// TwinCAT 3 PLC project PLC
// ProgramVersion: 3.1.4024.0
// libraries:
//   EfficientIO Energy Basic, * (EfficientIO)
//   Lynus Persistent Data V1, * (Lynus AG)
//   Lynus Standards, * (EfficientIO)
//   Tc2_EtherCAT, * (Beckhoff Automation GmbH)
//   Tc2_Standard, * (Beckhoff Automation GmbH)
//   Tc2_System, * (Beckhoff Automation GmbH)
//   Tc2_Utilities, * (Beckhoff Automation GmbH)
//   Tc3_Module, * (Beckhoff Automation GmbH)
// project tree:
//   FBs/EL3443_DPM/DUTs/ E_EL3443_DPM_Phase.TcDUT (not stored), E_EL3443_DPM_Total.TcDUT (not stored), MDP5001_341_7CD731EE.TcDUT (not stored), MDP5001_341_I_7CD731EE.TcDUT (not stored), MDP5001_341_O_7CD731EE.TcDUT (not stored), ST_EL3443_DPM_MUX_REAL.TcDUT (not stored), ST_EL3443_DPM_MUX_ULINT.TcDUT (not stored), ST_EL3443_DPM_StatusLx.TcDUT (not stored), ST_EL3443_DPM_StatusTotal.TcDUT (not stored), ST_EL3443_DPM_VariantLx.TcDUT (not stored), ST_EL3443_DPM_VariantTotal.TcDUT (not stored), ST_EL3443_DPM_VariantValues.TcDUT (not stored)
//   FBs/EL3443_DPM/ FB_EL3443_DPM.TcPOU (not stored)
//   FBs/EL3446 FW02 or higher/DUTs/ E_EL3446_Phase.TcDUT (not stored), MDP5001_342_066CA8C6.TcDUT (not stored), MDP5001_342_I_066CA8C6.TcDUT (not stored), MDP5001_342_O_066CA8C6.TcDUT (not stored), ST_EL3446_MUX_REAL.TcDUT, ST_EL3446_MUX_ULINT.TcDUT (not stored), ST_EL3446_StatusIx.TcDUT (not stored), ST_EL3446_VariantIx.TcDUT (not stored), ST_EL3446_VariantValues.TcDUT (not stored)
//   FBs/EL3446 FW02 or higher/ FB_EL3446.TcPOU (not stored)
//   FBs/ FB_CoE_EL3443.TcPOU (not stored), FB_CoE_EL3446.TcPOU (not stored), FB_EM_Beckhoff_EL3443.TcPOU (not stored), FB_EM_Beckhoff_EL3446.TcPOU (not stored)
//   / PlcTask.TcTTO
//   POUs/ prgEM.TcPOU, prgHW.TcPOU
// real-time tasks:
//   TASK PlcTask: cycle T#10ms, priority 20, ADS port 350
// I/O:
//   DEVICE Gerät 2 (EtherCAT), AmsNetId 5.146.125.98.3.1
//     Klemme 1 (EK1200) [EK1200-5000 EtherCAT Netzteil (2A E-Bus)]
//       Klemme 2 (EL3443) [EL3443 3K. Leistungsmessung]
//       Klemme 3 (EL3446) [EL3446 DPM 6 K. Strommessklemme]
//       Klemme 4 (EL3446) [EL3446 DPM 6 K. Strommessklemme]
//       Klemme 5 (EL9011) [EL9011 Endklemme]
// variable links:
//   PLC/PLC Instance <-> Device 2 (EtherCAT)/Term 1 (EK1200)/Term 2 (EL3443)
//     PlcTask Inputs/prgHW.MDP5001_341_DPM_Data_Data_{1..20} <-> DPM Data/Data {1..20}  (20 links)
//     PlcTask Inputs/prgHW.MDP5001_341_L1_Basic_Current <-> L1 Basic/Current
//     PlcTask Inputs/prgHW.MDP5001_341_L2_Basic_Current <-> L2 Basic/Current
//     PlcTask Inputs/prgHW.MDP5001_341_L3_Basic_Current <-> L3 Basic/Current
//     PlcTask Inputs/prgHW.MDP5001_341_L1_Basic_Voltage <-> L1 Basic/Voltage
//     PlcTask Inputs/prgHW.MDP5001_341_L2_Basic_Voltage <-> L2 Basic/Voltage
//     PlcTask Inputs/prgHW.MDP5001_341_L3_Basic_Voltage <-> L3 Basic/Voltage
//     PlcTask Inputs/prgHW.MDP5001_341_L1_Power_Active_Power <-> L1 Power/Active Power
//     PlcTask Inputs/prgHW.MDP5001_341_L2_Power_Active_Power <-> L2 Power/Active Power
//     PlcTask Inputs/prgHW.MDP5001_341_L3_Power_Active_Power <-> L3 Power/Active Power
//     PlcTask Inputs/prgHW.MDP5001_341_L1_Power_Apparent_Power <-> L1 Power/Apparent Power
//     PlcTask Inputs/prgHW.MDP5001_341_L2_Power_Apparent_Power <-> L2 Power/Apparent Power
//     PlcTask Inputs/prgHW.MDP5001_341_L3_Power_Apparent_Power <-> L3 Power/Apparent Power
//     PlcTask Inputs/prgHW.MDP5001_341_L1_Power_Power_Factor <-> L1 Power/Power Factor
//     PlcTask Inputs/prgHW.MDP5001_341_L2_Power_Power_Factor <-> L2 Power/Power Factor
//     PlcTask Inputs/prgHW.MDP5001_341_L3_Power_Power_Factor <-> L3 Power/Power Factor
//     PlcTask Inputs/prgHW.MDP5001_341_L1_Power_Reactive_Power <-> L1 Power/Reactive Power
//     PlcTask Inputs/prgHW.MDP5001_341_L2_Power_Reactive_Power <-> L2 Power/Reactive Power
//     PlcTask Inputs/prgHW.MDP5001_341_L3_Power_Reactive_Power <-> L3 Power/Reactive Power
//     PlcTask Inputs/prgHW.MDP5001_341_L1_Status_Current_Guard_Error <-> L1 Status/Current Guard Error
//     PlcTask Inputs/prgHW.MDP5001_341_L2_Status_Current_Guard_Error <-> L2 Status/Current Guard Error
//     PlcTask Inputs/prgHW.MDP5001_341_L3_Status_Current_Guard_Error <-> L3 Status/Current Guard Error
//     PlcTask Inputs/prgHW.MDP5001_341_L1_Status_Current_Guard_Warning <-> L1 Status/Current Guard Warning
//     PlcTask Inputs/prgHW.MDP5001_341_L2_Status_Current_Guard_Warning <-> L2 Status/Current Guard Warning
//     PlcTask Inputs/prgHW.MDP5001_341_L3_Status_Current_Guard_Warning <-> L3 Status/Current Guard Warning
//     PlcTask Inputs/prgHW.MDP5001_341_L1_Status_Inaccurate_Current <-> L1 Status/Inaccurate Current
//     PlcTask Inputs/prgHW.MDP5001_341_L2_Status_Inaccurate_Current <-> L2 Status/Inaccurate Current
//     PlcTask Inputs/prgHW.MDP5001_341_L3_Status_Inaccurate_Current <-> L3 Status/Inaccurate Current
//     PlcTask Inputs/prgHW.MDP5001_341_L1_Status_Inaccurate_Voltage <-> L1 Status/Inaccurate Voltage
//     PlcTask Inputs/prgHW.MDP5001_341_L2_Status_Inaccurate_Voltage <-> L2 Status/Inaccurate Voltage
//     PlcTask Inputs/prgHW.MDP5001_341_L3_Status_Inaccurate_Voltage <-> L3 Status/Inaccurate Voltage
//     PlcTask Inputs/prgHW.MDP5001_341_L1_Status_Overcurrent <-> L1 Status/Overcurrent
//     PlcTask Inputs/prgHW.MDP5001_341_L2_Status_Overcurrent <-> L2 Status/Overcurrent
//     PlcTask Inputs/prgHW.MDP5001_341_L3_Status_Overcurrent <-> L3 Status/Overcurrent
//     PlcTask Inputs/prgHW.MDP5001_341_L1_Status_Overvoltage <-> L1 Status/Overvoltage
//     PlcTask Inputs/prgHW.MDP5001_341_L2_Status_Overvoltage <-> L2 Status/Overvoltage
//     PlcTask Inputs/prgHW.MDP5001_341_L3_Status_Overvoltage <-> L3 Status/Overvoltage
//     PlcTask Inputs/prgHW.MDP5001_341_L1_Status_TxPDO_Toggle <-> L1 Status/TxPDO Toggle
//     PlcTask Inputs/prgHW.MDP5001_341_L2_Status_TxPDO_Toggle <-> L2 Status/TxPDO Toggle
//     PlcTask Inputs/prgHW.MDP5001_341_L3_Status_TxPDO_Toggle <-> L3 Status/TxPDO Toggle
//     PlcTask Inputs/prgHW.MDP5001_341_L1_Status_Voltage_Guard_Error <-> L1 Status/Voltage Guard Error
//     PlcTask Inputs/prgHW.MDP5001_341_L2_Status_Voltage_Guard_Error <-> L2 Status/Voltage Guard Error
//     PlcTask Inputs/prgHW.MDP5001_341_L3_Status_Voltage_Guard_Error <-> L3 Status/Voltage Guard Error
//     PlcTask Inputs/prgHW.MDP5001_341_L1_Status_Voltage_Guard_Warning <-> L1 Status/Voltage Guard Warning
//     PlcTask Inputs/prgHW.MDP5001_341_L2_Status_Voltage_Guard_Warning <-> L2 Status/Voltage Guard Warning
//     PlcTask Inputs/prgHW.MDP5001_341_L3_Status_Voltage_Guard_Warning <-> L3 Status/Voltage Guard Warning
//     PlcTask Inputs/prgHW.MDP5001_341_L1_Status_Voltage_Sign_Bit <-> L1 Status/Voltage Sign Bit
//     PlcTask Inputs/prgHW.MDP5001_341_L2_Status_Voltage_Sign_Bit <-> L2 Status/Voltage Sign Bit
//     PlcTask Inputs/prgHW.MDP5001_341_L3_Status_Voltage_Sign_Bit <-> L3 Status/Voltage Sign Bit
//     PlcTask Inputs/prgHW.MDP5001_341_Total_Basic_Calculated_Neutral_Line_Current <-> Total Basic/Calculated Neutral Line Current
//     PlcTask Inputs/prgHW.MDP5001_341_Total_Basic_Frequency <-> Total Basic/Frequency
//     PlcTask Inputs/prgHW.MDP5001_341_Total_Basic_Power_Factor <-> Total Basic/Power Factor
//     PlcTask Inputs/prgHW.MDP5001_341_Total_Status_Active_Power_Guard_Error <-> Total Status/Active Power Guard Error
//     PlcTask Inputs/prgHW.MDP5001_341_Total_Status_Active_Power_Guard_Warning <-> Total Status/Active Power Guard Warning
//     PlcTask Inputs/prgHW.MDP5001_341_Total_Status_Apparent_Power_Guard_Error <-> Total Status/Apparent Power Guard Error
//     PlcTask Inputs/prgHW.MDP5001_341_Total_Status_Apparent_Power_Guard_Warning <-> Total Status/Apparent Power Guard Warning
//     PlcTask Inputs/prgHW.MDP5001_341_Total_Status_Frequency_Guard_Error <-> Total Status/Frequency Guard Error
//     PlcTask Inputs/prgHW.MDP5001_341_Total_Status_Frequency_Guard_Warning <-> Total Status/Frequency Guard Warning
//     PlcTask Inputs/prgHW.MDP5001_341_Total_Status_Grid_Direction <-> Total Status/Grid Direction
//     PlcTask Inputs/prgHW.MDP5001_341_Total_Status_Neutral_Current_Guard_Error <-> Total Status/Neutral Current Guard Error
//     PlcTask Inputs/prgHW.MDP5001_341_Total_Status_Neutral_Current_Guard_Warning <-> Total Status/Neutral Current Guard Warning
//     PlcTask Inputs/prgHW.MDP5001_341_Total_Status_Power_Quality_Factor <-> Total Status/Power Quality Factor
//     PlcTask Inputs/prgHW.MDP5001_341_Total_Status_Power_Quality_Guard_Error <-> Total Status/Power Quality Guard Error
//     PlcTask Inputs/prgHW.MDP5001_341_Total_Status_Power_Quality_Guard_Warning <-> Total Status/Power Quality Guard Warning
//     PlcTask Inputs/prgHW.MDP5001_341_Total_Status_System_State <-> Total Status/System State
//     PlcTask Inputs/prgHW.MDP5001_341_Total_Status_TxPDO_State <-> Total Status/TxPDO State
//     PlcTask Inputs/prgHW.MDP5001_341_Total_Status_TxPDO_Toggle <-> Total Status/TxPDO Toggle
//     PlcTask Inputs/prgHW.MDP5001_341_Total_Variant_Value_In_Index_1_REAL <-> Total Variant Value In/Index 1 REAL
//     PlcTask Inputs/prgHW.MDP5001_341_Total_Variant_Value_In_Index_2_REAL <-> Total Variant Value In/Index 2 REAL
//     PlcTask Inputs/prgHW.MDP5001_341_Total_Variant_Value_In_Index_3_REAL <-> Total Variant Value In/Index 3 REAL
//     PlcTask Inputs/prgHW.MDP5001_341_Total_Variant_Value_In_Index_4_ULINT <-> Total Variant Value In/Index 4 ULINT
//     PlcTask Inputs/prgHW.MDP5001_341_Total_Variant_Value_In_TxPDO_Toggle <-> Total Variant Value In/TxPDO Toggle
//     PlcTask Inputs/prgHW.MDP5001_341_Total_Variant_Value_In_Value_1_REAL <-> Total Variant Value In/Value 1 REAL
//     PlcTask Inputs/prgHW.MDP5001_341_Total_Variant_Value_In_Value_2_REAL <-> Total Variant Value In/Value 2 REAL
//     PlcTask Inputs/prgHW.MDP5001_341_Total_Variant_Value_In_Value_3_REAL <-> Total Variant Value In/Value 3 REAL
//     PlcTask Inputs/prgHW.MDP5001_341_Total_Variant_Value_In_Value_4_ULINT <-> Total Variant Value In/Value 4 ULINT
//     PlcTask Outputs/prgHW.MDP5001_341_Total_Interval_Reset_Interval <-> Total Interval/Reset Interval
//     PlcTask Outputs/prgHW.MDP5001_341_Total_Variant_Value_Out_Index_1_REAL <-> Total Variant Value Out/Index 1 REAL
//     PlcTask Outputs/prgHW.MDP5001_341_Total_Variant_Value_Out_Index_2_REAL <-> Total Variant Value Out/Index 2 REAL
//     PlcTask Outputs/prgHW.MDP5001_341_Total_Variant_Value_Out_Index_3_REAL <-> Total Variant Value Out/Index 3 REAL
//     PlcTask Outputs/prgHW.MDP5001_341_Total_Variant_Value_Out_Index_4_ULINT <-> Total Variant Value Out/Index 4 ULINT
//   PLC/PLC Instance <-> Device 2 (EtherCAT)/Term 1 (EK1200)/Term 3 (EL3446)
//     PlcTask Inputs/prgHW.MDP5001_342_DPM_Variant_Value_In_Index_1_REAL_1 <-> DPM Variant Value In/Index 1 REAL
//     PlcTask Inputs/prgHW.MDP5001_342_DPM_Variant_Value_In_Index_2_REAL_1 <-> DPM Variant Value In/Index 2 REAL
//     PlcTask Inputs/prgHW.MDP5001_342_DPM_Variant_Value_In_Index_3_REAL_1 <-> DPM Variant Value In/Index 3 REAL
//     PlcTask Inputs/prgHW.MDP5001_342_DPM_Variant_Value_In_Index_4_ULINT_1 <-> DPM Variant Value In/Index 4 ULINT
//     PlcTask Inputs/prgHW.MDP5001_342_DPM_Variant_Value_In_TxPDO_Toggle_1 <-> DPM Variant Value In/TxPDO Toggle
//     PlcTask Inputs/prgHW.MDP5001_342_DPM_Variant_Value_In_Value_1_REAL_1 <-> DPM Variant Value In/Value 1 REAL
//     PlcTask Inputs/prgHW.MDP5001_342_DPM_Variant_Value_In_Value_2_REAL_1 <-> DPM Variant Value In/Value 2 REAL
//     PlcTask Inputs/prgHW.MDP5001_342_DPM_Variant_Value_In_Value_3_REAL_1 <-> DPM Variant Value In/Value 3 REAL
//     PlcTask Inputs/prgHW.MDP5001_342_DPM_Variant_Value_In_Value_4_ULINT_1 <-> DPM Variant Value In/Value 4 ULINT
//     PlcTask Inputs/prgHW.MDP5001_342_I{1..6}_Channel_Active_Energy_1 <-> I{1..6} Channel/Active Energy  (6 links)
//     PlcTask Inputs/prgHW.MDP5001_342_I{1..6}_Channel_Active_Power_1 <-> I{1..6} Channel/Active Power  (6 links)
//     PlcTask Inputs/prgHW.MDP5001_342_I{1..6}_Channel_Active_Power_Guard_Error_1 <-> I{1..6} Channel/Active Power Guard Error  (6 links)
//     PlcTask Inputs/prgHW.MDP5001_342_I{1..6}_Channel_Active_Power_Guard_Warning_1 <-> I{1..6} Channel/Active Power Guard Warning  (6 links)
//     PlcTask Inputs/prgHW.MDP5001_342_I{1..6}_Channel_Apparent_Power_1 <-> I{1..6} Channel/Apparent Power  (6 links)
//     PlcTask Inputs/prgHW.MDP5001_342_I{1..6}_Channel_Apparent_Power_Guard_Error_1 <-> I{1..6} Channel/Apparent Power Guard Error  (6 links)
//     PlcTask Inputs/prgHW.MDP5001_342_I{1..6}_Channel_Apparent_Power_Guard_Warning_1 <-> I{1..6} Channel/Apparent Power Guard Warning  (6 links)
//     PlcTask Inputs/prgHW.MDP5001_342_I{1..6}_Channel_Current_1 <-> I{1..6} Channel/Current  (6 links)
//     PlcTask Inputs/prgHW.MDP5001_342_I{1..6}_Channel_Current_Guard_Error_1 <-> I{1..6} Channel/Current Guard Error  (6 links)
//     PlcTask Inputs/prgHW.MDP5001_342_I{1..6}_Channel_Current_Guard_Warning_1 <-> I{1..6} Channel/Current Guard Warning  (6 links)
//     PlcTask Inputs/prgHW.MDP5001_342_I{1..6}_Channel_DPM_Inaccurate_1 <-> I{1..6} Channel/DPM Inaccurate  (6 links)
//     PlcTask Inputs/prgHW.MDP5001_342_I{1..6}_Channel_DPM_Timeout_1 <-> I{1..6} Channel/DPM Timeout  (6 links)
//     PlcTask Inputs/prgHW.MDP5001_342_I{1..6}_Channel_Inaccurate_Current_1 <-> I{1..6} Channel/Inaccurate Current  (6 links)
//     PlcTask Inputs/prgHW.MDP5001_342_I{1..6}_Channel_Overcurrent_1 <-> I{1..6} Channel/Overcurrent  (6 links)
//     PlcTask Inputs/prgHW.MDP5001_342_I{1..6}_Channel_Reactive_Power_Fundamental_1 <-> I{1..6} Channel/Reactive Power Fundamental  (6 links)
//     PlcTask Inputs/prgHW.MDP5001_342_I{1..6}_Channel_Reactive_Power_Guard_Error_1 <-> I{1..6} Channel/Reactive Power Guard Error  (6 links)
//     PlcTask Inputs/prgHW.MDP5001_342_I{1..6}_Channel_Reactive_Power_Guard_Warning_1 <-> I{1..6} Channel/Reactive Power Guard Warning  (6 links)
//     PlcTask Inputs/prgHW.MDP5001_342_I{1..6}_Channel_TxPDO_Toggle_1 <-> I{1..6} Channel/TxPDO Toggle  (6 links)
//     PlcTask Outputs/prgHW.MDP5001_342_DPM_Data_Data_{1..20}_1 <-> DPM Data/Data {1..20}  (20 links)
//     PlcTask Outputs/prgHW.MDP5001_342_DPM_Variant_Value_Out_Index_1_REAL_1 <-> DPM Variant Value Out/Index 1 REAL
//     PlcTask Outputs/prgHW.MDP5001_342_DPM_Variant_Value_Out_Index_2_REAL_1 <-> DPM Variant Value Out/Index 2 REAL
//     PlcTask Outputs/prgHW.MDP5001_342_DPM_Variant_Value_Out_Index_3_REAL_1 <-> DPM Variant Value Out/Index 3 REAL
//     PlcTask Outputs/prgHW.MDP5001_342_DPM_Variant_Value_Out_Index_4_ULINT_1 <-> DPM Variant Value Out/Index 4 ULINT
//   PLC/PLC Instance <-> Device 2 (EtherCAT)/Term 1 (EK1200)/Term 4 (EL3446)
//     PlcTask Inputs/prgHW.MDP5001_342_DPM_Variant_Value_In_Index_1_REAL_2 <-> DPM Variant Value In/Index 1 REAL
//     PlcTask Inputs/prgHW.MDP5001_342_DPM_Variant_Value_In_Index_2_REAL_2 <-> DPM Variant Value In/Index 2 REAL
//     PlcTask Inputs/prgHW.MDP5001_342_DPM_Variant_Value_In_Index_3_REAL_2 <-> DPM Variant Value In/Index 3 REAL
//     PlcTask Inputs/prgHW.MDP5001_342_DPM_Variant_Value_In_Index_4_ULINT_2 <-> DPM Variant Value In/Index 4 ULINT
//     PlcTask Inputs/prgHW.MDP5001_342_DPM_Variant_Value_In_TxPDO_Toggle_2 <-> DPM Variant Value In/TxPDO Toggle
//     PlcTask Inputs/prgHW.MDP5001_342_DPM_Variant_Value_In_Value_1_REAL_2 <-> DPM Variant Value In/Value 1 REAL
//     PlcTask Inputs/prgHW.MDP5001_342_DPM_Variant_Value_In_Value_2_REAL_2 <-> DPM Variant Value In/Value 2 REAL
//     PlcTask Inputs/prgHW.MDP5001_342_DPM_Variant_Value_In_Value_3_REAL_2 <-> DPM Variant Value In/Value 3 REAL
//     PlcTask Inputs/prgHW.MDP5001_342_DPM_Variant_Value_In_Value_4_ULINT_2 <-> DPM Variant Value In/Value 4 ULINT
//     PlcTask Inputs/prgHW.MDP5001_342_I{1..6}_Channel_Active_Energy_2 <-> I{1..6} Channel/Active Energy  (6 links)
//     PlcTask Inputs/prgHW.MDP5001_342_I{1..6}_Channel_Active_Power_2 <-> I{1..6} Channel/Active Power  (6 links)
//     PlcTask Inputs/prgHW.MDP5001_342_I{1..6}_Channel_Active_Power_Guard_Error_2 <-> I{1..6} Channel/Active Power Guard Error  (6 links)
//     PlcTask Inputs/prgHW.MDP5001_342_I{1..6}_Channel_Active_Power_Guard_Warning_2 <-> I{1..6} Channel/Active Power Guard Warning  (6 links)
//     PlcTask Inputs/prgHW.MDP5001_342_I{1..6}_Channel_Apparent_Power_2 <-> I{1..6} Channel/Apparent Power  (6 links)
//     PlcTask Inputs/prgHW.MDP5001_342_I{1..6}_Channel_Apparent_Power_Guard_Error_2 <-> I{1..6} Channel/Apparent Power Guard Error  (6 links)
//     PlcTask Inputs/prgHW.MDP5001_342_I{1..6}_Channel_Apparent_Power_Guard_Warning_2 <-> I{1..6} Channel/Apparent Power Guard Warning  (6 links)
//     PlcTask Inputs/prgHW.MDP5001_342_I{1..6}_Channel_Current_2 <-> I{1..6} Channel/Current  (6 links)
//     PlcTask Inputs/prgHW.MDP5001_342_I{1..6}_Channel_Current_Guard_Error_2 <-> I{1..6} Channel/Current Guard Error  (6 links)
//     PlcTask Inputs/prgHW.MDP5001_342_I{1..6}_Channel_Current_Guard_Warning_2 <-> I{1..6} Channel/Current Guard Warning  (6 links)
//     PlcTask Inputs/prgHW.MDP5001_342_I{1..6}_Channel_DPM_Inaccurate_2 <-> I{1..6} Channel/DPM Inaccurate  (6 links)
//     PlcTask Inputs/prgHW.MDP5001_342_I{1..6}_Channel_DPM_Timeout_2 <-> I{1..6} Channel/DPM Timeout  (6 links)
//     PlcTask Inputs/prgHW.MDP5001_342_I{1..6}_Channel_Inaccurate_Current_2 <-> I{1..6} Channel/Inaccurate Current  (6 links)
//     PlcTask Inputs/prgHW.MDP5001_342_I{1..6}_Channel_Overcurrent_2 <-> I{1..6} Channel/Overcurrent  (6 links)
//     PlcTask Inputs/prgHW.MDP5001_342_I{1..6}_Channel_Reactive_Power_Fundamental_2 <-> I{1..6} Channel/Reactive Power Fundamental  (6 links)
//     PlcTask Inputs/prgHW.MDP5001_342_I{1..6}_Channel_Reactive_Power_Guard_Error_2 <-> I{1..6} Channel/Reactive Power Guard Error  (6 links)
//     PlcTask Inputs/prgHW.MDP5001_342_I{1..6}_Channel_Reactive_Power_Guard_Warning_2 <-> I{1..6} Channel/Reactive Power Guard Warning  (6 links)
//     PlcTask Inputs/prgHW.MDP5001_342_I{1..6}_Channel_TxPDO_Toggle_2 <-> I{1..6} Channel/TxPDO Toggle  (6 links)
//     PlcTask Outputs/prgHW.MDP5001_342_DPM_Data_Data_{1..20}_2 <-> DPM Data/Data {1..20}  (20 links)
//     PlcTask Outputs/prgHW.MDP5001_342_DPM_Variant_Value_Out_Index_1_REAL_2 <-> DPM Variant Value Out/Index 1 REAL
//     PlcTask Outputs/prgHW.MDP5001_342_DPM_Variant_Value_Out_Index_2_REAL_2 <-> DPM Variant Value Out/Index 2 REAL
//     PlcTask Outputs/prgHW.MDP5001_342_DPM_Variant_Value_Out_Index_3_REAL_2 <-> DPM Variant Value Out/Index 3 REAL
//     PlcTask Outputs/prgHW.MDP5001_342_DPM_Variant_Value_Out_Index_4_ULINT_2 <-> DPM Variant Value Out/Index 4 ULINT

CONFIGURATION PLC
    RESOURCE PLC ON TwinCAT3
        TASK PlcTask(INTERVAL := T#10ms, PRIORITY := 20);
        PROGRAM prgEM WITH PlcTask : prgEM;
        PROGRAM prgHW WITH PlcTask : prgHW;
    END_RESOURCE
END_CONFIGURATION

// ---- FBs/EL3446 FW02 or higher/DUTs/ST_EL3446_MUX_REAL.TcDUT
TYPE ST_EL3446_MUX_REAL :
STRUCT
    nSelector : UINT := E_EL3446_Phase.Error_INDEX_Not_Valid;
    fValueRef : REFERENCE TO REAL;
END_STRUCT
END_TYPE

// ---- POUs/prgEM.TcPOU
PROGRAM prgEM
VAR
	fbEL3443DPM 		: FB_EM_Beckhoff_EL3443;	//EL3443 | PDO Assignment "DPM" (DPM: Distributed Power Measurement) |3-phase power measurement terminal with extended functionality
	fb_EL3446_1			: FB_EM_Beckhoff_EL3446;
	fb_EL3446_2			: FB_EM_Beckhoff_EL3446;
	lr_RealPower_Halle	: LREAL;						
	lr_ApparentPower_Halle: LREAL;						
	lr_ReactivePower_Halle: LREAL;						
	lr_Frequency_Halle	: LREAL;						
                                                        
	lr_Voltage_L1N		: LREAL;						
	lr_Voltage_L2N		: LREAL;						
	lr_Voltage_L3N		: LREAL;						
	lr_Voltage_L1L2		: LREAL;						
	lr_Voltage_L2L3		: LREAL;						
	lr_Voltage_L3L1		: LREAL;						
 	lr_Current_L1		: LREAL;						
	lr_Current_L2		: LREAL;						
	lr_Current_L3		: LREAL;						

	lr_RealPower_Hundegger	: LREAL;						
	lr_RealPower_Spannex	: LREAL;		
	lr_RealPower_Kran		: LREAL;	
	real_Array_Modbus_Data	AT%MB0 : ARRAY[0..49] OF REAL;
	
END_VAR
VAR_INPUT
	stEL3443_IO 						: MDP5001_341_7CD731EE;
	stEL3446_IO_1 						: MDP5001_342_066CA8C6; 
	stEL3446_IO_2 						: MDP5001_342_066CA8C6; 
END_VAR
VAR PERSISTENT
	lr_EnergyCounter_Halle	: LREAL;						
END_VAR

// grid measurement
fbEL3443DPM(
	bEnable 	:= TRUE, 
	bInvers_CH1 := FALSE, 
	bInvers_CH2	:= FALSE, 
	bInvers_CH3	:= FALSE, 
	uiCurrentTransformerRatio:= 300,		// two cables,300:1 CTs only over one cable 
	nSlaveAddr 	:= 1001,
	b_SubIndex	:= 2,
	stEL3443_IO := ,
	pDpmData=> , 
	stDataEMPower=> , 
	stDataEMCounter=> , 
	stDataEMPowerRealTime=> , 
	stDataEMCounterRealTime=> );
fbEL3443DPM.stEL3443_IO.MDP5001_341_Input := stEL3443_IO.MDP5001_341_Input;
stEL3443_IO.MDP5001_341_Output	:= fbEL3443DPM.stEL3443_IO.MDP5001_341_Output;
 	
lr_RealPower_Halle 		:= fbEL3443DPM.stDataEMPower.lrPowerTotal; 	
lr_ApparentPower_Halle 	:= fbEL3443DPM.stDataEMPower.lrApparentPowerTotal;
lr_ReactivePower_Halle	:= fbEL3443DPM.stDataEMPower.lrReactivePowerTotal;
lr_Frequency_Halle		:= fbEL3443DPM.stDataEMPower.lrFrequency;
lr_Voltage_L1N			:= fbEL3443DPM.stDataEMPower.lrVoltageL1N;
lr_Voltage_L2N			:= fbEL3443DPM.stDataEMPower.lrVoltageL2N;
lr_Voltage_L3N			:= fbEL3443DPM.stDataEMPower.lrVoltageL3N;
lr_Voltage_L1L2			:= fbEL3443DPM.stDataEMPower.lrVoltageL1L2;
lr_Voltage_L2L3			:= fbEL3443DPM.stDataEMPower.lrVoltageL2L3;
lr_Voltage_L3L1			:= fbEL3443DPM.stDataEMPower.lrVoltageL3L1;
lr_EnergyCounter_Halle	:= fbEL3443DPM.stDataEMCounter.lrTotalCounterEnergy_Consumption;
lr_Current_L1			:= fbEL3443DPM.stDataEMPower.lrCurrentL1;
lr_Current_L2			:= fbEL3443DPM.stDataEMPower.lrCurrentL2;
lr_Current_L3			:= fbEL3443DPM.stDataEMPower.lrCurrentL3;
	 
fb_EL3446_1(
	bEnable:= TRUE , 
	bEnableVariantValues:= TRUE, 
	pDpmData:= fbEL3443DPM.pDpmData, 
	nSlaveAddr:= 1002, 
	b_SubIndex	:= 2,
	bInvers_CH1:= FALSE, 
	bInvers_CH2:= FALSE, 
	bInvers_CH3:= FALSE, 
	bInvers_CH4:= FALSE, 
	bInvers_CH5:= FALSE, 
	bInvers_CH6:= FALSE, 
	uiCurrentTransformerRatio_CH1:= 300, 
	uiCurrentTransformerRatio_CH2:= 300, 
	uiCurrentTransformerRatio_CH3:= 300, 
	uiCurrentTransformerRatio_CH4:= 300, 
	uiCurrentTransformerRatio_CH5:= 300, 
	uiCurrentTransformerRatio_CH6:= 300, 
	uiVoltagePhaseSelector_CH1:= , 
	uiVoltagePhaseSelector_CH2:= , 
	uiVoltagePhaseSelector_CH3:= , 
	uiVoltagePhaseSelector_CH4:= , 
	uiVoltagePhaseSelector_CH5:= , 
	uiVoltagePhaseSelector_CH6:= , 
	bEnable3PhaseCH13:= , 
	bEnable3PhaseCH46:= , 
	stDataEMPowerRealTime:= fbEL3443DPM.stDataEMPowerRealTime, 
	stEL3446_IO := ,
	stDataEMPower_CH1=> , 
	stDataEMCounter_CH1=> , 
	stDataEMPowerRealTime_CH1=> , 
	stDataEMCounterRealTime_CH1=> , 
	stDataEMPower_CH2=> , 
	stDataEMCounter_CH2=> , 
	stDataEMPowerRealTime_CH2=> , 
	stDataEMCounterRealTime_CH2=> , 
	stDataEMPower_CH3=> , 
	stDataEMCounter_CH3=> , 
	stDataEMPowerRealTime_CH3=> , 
	stDataEMCounterRealTime_CH3=> , 
	stDataEMPower_CH4=> , 
	stDataEMCounter_CH4=> , 
	stDataEMPowerRealTime_CH4=> , 
	stDataEMCounterRealTime_CH4=> , 
	stDataEMPower_CH5=> , 
	stDataEMCounter_CH5=> , 
	stDataEMPowerRealTime_CH5=> , 
	stDataEMCounterRealTime_CH5=> , 
	stDataEMPower_CH6=> , 
	stDataEMCounter_CH6=> , 
	stDataEMPowerRealTime_CH6=> , 
	stDataEMCounterRealTime_CH6=> );
fb_EL3446_1.stEL3446_IO.MDP5001_342_Input := stEL3446_IO_1.MDP5001_342_Input;
stEL3446_IO_1.MDP5001_342_Output := 	fb_EL3446_1.stEL3446_IO.MDP5001_342_Output;


fb_EL3446_2(
	bEnable:= TRUE , 
	bEnableVariantValues:= TRUE, 
	pDpmData:= fbEL3443DPM.pDpmData, 
	nSlaveAddr:= 1003, 
	b_SubIndex	:= 2,
	bInvers_CH1:= TRUE, 
	bInvers_CH2:= TRUE, 
	bInvers_CH3:= TRUE, 
	bInvers_CH4:= TRUE, 
	bInvers_CH5:= TRUE, 
	bInvers_CH6:= TRUE,	
	uiCurrentTransformerRatio_CH1:= 300, 
	uiCurrentTransformerRatio_CH2:= 300, 
	uiCurrentTransformerRatio_CH3:= 300, 
	uiCurrentTransformerRatio_CH4:= 300, 
	uiCurrentTransformerRatio_CH5:= 300, 
	uiCurrentTransformerRatio_CH6:= 300, 
	uiVoltagePhaseSelector_CH1:= , 
	uiVoltagePhaseSelector_CH2:= , 
	uiVoltagePhaseSelector_CH3:= , 
	uiVoltagePhaseSelector_CH4:= , 
	uiVoltagePhaseSelector_CH5:= , 
	uiVoltagePhaseSelector_CH6:= , 
	bEnable3PhaseCH13:= TRUE, 
	bEnable3PhaseCH46:= TRUE, 
	stDataEMPowerRealTime:= fbEL3443DPM.stDataEMPowerRealTime, 
	stEL3446_IO := ,
	stDataEMPower_CH1=> , 
	stDataEMCounter_CH1=> , 
	stDataEMPowerRealTime_CH1=> , 
	stDataEMCounterRealTime_CH1=> , 
	stDataEMPower_CH2=> , 
	stDataEMCounter_CH2=> , 
	stDataEMPowerRealTime_CH2=> , 
	stDataEMCounterRealTime_CH2=> , 
	stDataEMPower_CH3=> , 
	stDataEMCounter_CH3=> , 
	stDataEMPowerRealTime_CH3=> , 
	stDataEMCounterRealTime_CH3=> , 
	stDataEMPower_CH4=> , 
	stDataEMCounter_CH4=> , 
	stDataEMPowerRealTime_CH4=> , 
	stDataEMCounterRealTime_CH4=> , 
	stDataEMPower_CH5=> , 
	stDataEMCounter_CH5=> , 
	stDataEMPowerRealTime_CH5=> , 
	stDataEMCounterRealTime_CH5=> , 
	stDataEMPower_CH6=> , 
	stDataEMCounter_CH6=> , 
	stDataEMPowerRealTime_CH6=> , 
	stDataEMCounterRealTime_CH6=> );
fb_EL3446_2.stEL3446_IO.MDP5001_342_Input := stEL3446_IO_2.MDP5001_342_Input;
stEL3446_IO_2.MDP5001_342_Output := 	fb_EL3446_2.stEL3446_IO.MDP5001_342_Output;

lr_RealPower_Hundegger	:= fb_EL3446_1.stDataEMPower_CH1.lrPowerConsumption;
lr_RealPower_Spannex	:= fb_EL3446_1.stDataEMPower_CH4.lrPowerConsumption;
lr_RealPower_Kran		:= fb_EL3446_2.stDataEMPower_CH1.lrPowerConsumption;

real_Array_Modbus_Data[0] 	:= 		 INT_TO_REAL(REAL_TO_INT(LREAL_TO_REAL(lr_RealPower_Halle     	*10)))/10 ;
real_Array_Modbus_Data[1] 	:= 		 INT_TO_REAL(REAL_TO_INT(LREAL_TO_REAL(lr_ApparentPower_Halle  	*10)))/10 ;
real_Array_Modbus_Data[2] 	:= 		 INT_TO_REAL(REAL_TO_INT(LREAL_TO_REAL(lr_ReactivePower_Halle  	*10)))/10 ;
real_Array_Modbus_Data[3] 	:= 		 INT_TO_REAL(REAL_TO_INT(LREAL_TO_REAL(lr_Frequency_Halle 		*10)))/10 ;
real_Array_Modbus_Data[4] 	:= 		 INT_TO_REAL(REAL_TO_INT(LREAL_TO_REAL(lr_Voltage_L1N  			*10)))/10 ;
real_Array_Modbus_Data[5] 	:= 		 INT_TO_REAL(REAL_TO_INT(LREAL_TO_REAL(lr_Voltage_L2N  			*10)))/10 ;
real_Array_Modbus_Data[6] 	:= 		 INT_TO_REAL(REAL_TO_INT(LREAL_TO_REAL(lr_Voltage_L3N  			*10)))/10 ;
real_Array_Modbus_Data[7]	:=       INT_TO_REAL(REAL_TO_INT(LREAL_TO_REAL(lr_Voltage_L1L2			*10)))/10  ;
real_Array_Modbus_Data[8]	:=       INT_TO_REAL(REAL_TO_INT(LREAL_TO_REAL(lr_Voltage_L2L3			*10)))/10  ;
real_Array_Modbus_Data[9]	:=       INT_TO_REAL(REAL_TO_INT(LREAL_TO_REAL(lr_Voltage_L3L1			*10)))/10  ;
real_Array_Modbus_Data[10]	:=       INT_TO_REAL(REAL_TO_INT(LREAL_TO_REAL(lr_Current_L1			*10)))/10      ;
real_Array_Modbus_Data[11]	:=       INT_TO_REAL(REAL_TO_INT(LREAL_TO_REAL(lr_Current_L2			*10)))/10      ;
real_Array_Modbus_Data[12]	:=       INT_TO_REAL(REAL_TO_INT(LREAL_TO_REAL(lr_Current_L3			*10)))/10      ;
real_Array_Modbus_Data[13]	:=       INT_TO_REAL(REAL_TO_INT(LREAL_TO_REAL(lr_RealPower_Hundegger 	*10)))/10    ;
real_Array_Modbus_Data[14]	:=       INT_TO_REAL(REAL_TO_INT(LREAL_TO_REAL(lr_RealPower_Spannex  	*10)))/10    ;
real_Array_Modbus_Data[15]	:=       INT_TO_REAL(REAL_TO_INT(LREAL_TO_REAL(lr_RealPower_Kran		*10)))/10      ;

END_PROGRAM

// ---- POUs/prgHW.TcPOU
PROGRAM prgHW
VAR
	// IOs for EL3443
	{attribute 'TcLinkTo' := 'TIID^Gerät 2 (EtherCAT)^Klemme 1 (EK1200)^Klemme 2 (EL3443)^L1 Status^Voltage Sign Bit'}
	MDP5001_341_L1_Status_Voltage_Sign_Bit   	AT%I*  : BOOL;  // linked via attribute 
	{attribute 'TcLinkTo' := 'TIID^Gerät 2 (EtherCAT)^Klemme 1 (EK1200)^Klemme 2 (EL3443)^L1 Status^Overvoltage'}
	MDP5001_341_L1_Status_Overvoltage			AT%I*  : BOOL;  // linked via attribute 
	{attribute 'TcLinkTo' := 'TIID^Gerät 2 (EtherCAT)^Klemme 1 (EK1200)^Klemme 2 (EL3443)^L1 Status^Overcurrent'}
	MDP5001_341_L1_Status_Overcurrent			AT%I*  : BOOL;  // linked via attribute 
	{attribute 'TcLinkTo' := 'TIID^Gerät 2 (EtherCAT)^Klemme 1 (EK1200)^Klemme 2 (EL3443)^L1 Status^Inaccurate Voltage'}	
	MDP5001_341_L1_Status_Inaccurate_Voltage	AT%I*  : BOOL;  // linked via attribute 
	{attribute 'TcLinkTo' := 'TIID^Gerät 2 (EtherCAT)^Klemme 1 (EK1200)^Klemme 2 (EL3443)^L1 Status^Inaccurate Current'}
	MDP5001_341_L1_Status_Inaccurate_Current	AT%I*  : BOOL;  // linked via attribute 	
	{attribute 'TcLinkTo' := 'TIID^Gerät 2 (EtherCAT)^Klemme 1 (EK1200)^Klemme 2 (EL3443)^L1 Status^Voltage Guard Warning'}
	MDP5001_341_L1_Status_Voltage_Guard_Warning	AT%I*  : BOOL;  // linked via attribute
	{attribute 'TcLinkTo' := 'TIID^Gerät 2 (EtherCAT)^Klemme 1 (EK1200)^Klemme 2 (EL3443)^L1 Status^Voltage Guard Error'}
	MDP5001_341_L1_Status_Voltage_Guard_Error	AT%I*  : BOOL;  // linked via attribute
	{attribute 'TcLinkTo' := 'TIID^Gerät 2 (EtherCAT)^Klemme 1 (EK1200)^Klemme 2 (EL3443)^L1 Status^Current Guard Warning'}
	MDP5001_341_L1_Status_Current_Guard_Warning AT%I*  : BOOL;  // linked via attribute
	{attribute 'TcLinkTo' := 'TIID^Gerät 2 (EtherCAT)^Klemme 1 (EK1200)^Klemme 2 (EL3443)^L1 Status^Current Guard Error'}
	MDP5001_341_L1_Status_Current_Guard_Error	AT%I*  : BOOL;  // linked via attribute
	{attribute 'TcLinkTo' := 'TIID^Gerät 2 (EtherCAT)^Klemme 1 (EK1200)^Klemme 2 (EL3443)^L1 Status^TxPDO Toggle'}
	MDP5001_341_L1_Status_TxPDO_Toggle			AT%I*  : BOOL;  // linked via attribute
	{attribute 'TcLinkTo' := 'TIID^Gerät 2 (EtherCAT)^Klemme 1 (EK1200)^Klemme 2 (EL3443)^L1 Basic^Voltage'}
	MDP5001_341_L1_Basic_Voltage				AT%I*  : REAL;		// linked via attribute 
	{attribute 'TcLinkTo' := 'TIID^Gerät 2 (EtherCAT)^Klemme 1 (EK1200)^Klemme 2 (EL3443)^L1 Basic^Current'}
	MDP5001_341_L1_Basic_Current				AT%I*  : REAL;		// linked via attribute 
	{attribute 'TcLinkTo' := 'TIID^Gerät 2 (EtherCAT)^Klemme 1 (EK1200)^Klemme 2 (EL3443)^L1 Power^Active Power'}
	MDP5001_341_L1_Power_Active_Power			AT%I*  : REAL;		// linked via attribute 
	{attribute 'TcLinkTo' := 'TIID^Gerät 2 (EtherCAT)^Klemme 1 (EK1200)^Klemme 2 (EL3443)^L1 Power^Apparent Power'}
	MDP5001_341_L1_Power_Apparent_Power			AT%I* : REAL;		// linked via attribute 
	{attribute 'TcLinkTo' := 'TIID^Gerät 2 (EtherCAT)^Klemme 1 (EK1200)^Klemme 2 (EL3443)^L1 Power^Reactive Power'}
	MDP5001_341_L1_Power_Reactive_Power			AT%I* : REAL;		// linked via attribute 
	{attribute 'TcLinkTo' := 'TIID^Gerät 2 (EtherCAT)^Klemme 1 (EK1200)^Klemme 2 (EL3443)^L1 Power^Power Factor'}
	MDP5001_341_L1_Power_Power_Factor			AT%I* : REAL;		// linked via attribute 
	{attribute 'TcLinkTo' := 'TIID^Gerät 2 (EtherCAT)^Klemme 1 (EK1200)^Klemme 2 (EL3443)^L2 Status^Voltage Sign Bit'}
	MDP5001_341_L2_Status_Voltage_Sign_Bit   	AT%I*  : BOOL;  // linked via attribute 
	{attribute 'TcLinkTo' := 'TIID^Gerät 2 (EtherCAT)^Klemme 1 (EK1200)^Klemme 2 (EL3443)^L2 Status^Overvoltage'}
	MDP5001_341_L2_Status_Overvoltage			AT%I*  : BOOL;  // linked via attribute 
	{attribute 'TcLinkTo' := 'TIID^Gerät 2 (EtherCAT)^Klemme 1 (EK1200)^Klemme 2 (EL3443)^L2 Status^Overcurrent'}
	MDP5001_341_L2_Status_Overcurrent			AT%I*  : BOOL;  // linked via attribute 
	{attribute 'TcLinkTo' := 'TIID^Gerät 2 (EtherCAT)^Klemme 1 (EK1200)^Klemme 2 (EL3443)^L2 Status^Inaccurate Voltage'}	
	MDP5001_341_L2_Status_Inaccurate_Voltage	AT%I*  : BOOL;  // linked via attribute 
	{attribute 'TcLinkTo' := 'TIID^Gerät 2 (EtherCAT)^Klemme 1 (EK1200)^Klemme 2 (EL3443)^L2 Status^Inaccurate Current'}
	MDP5001_341_L2_Status_Inaccurate_Current	AT%I*  : BOOL;  // linked via attribute 	
	{attribute 'TcLinkTo' := 'TIID^Gerät 2 (EtherCAT)^Klemme 1 (EK1200)^Klemme 2 (EL3443)^L2 Status^Voltage Guard Warning'}
	MDP5001_341_L2_Status_Voltage_Guard_Warning	AT%I*  : BOOL;  // linked via attribute
	{attribute 'TcLinkTo' := 'TIID^Gerät 2 (EtherCAT)^Klemme 1 (EK1200)^Klemme 2 (EL3443)^L2 Status^Voltage Guard Error'}
	MDP5001_341_L2_Status_Voltage_Guard_Error	AT%I*  : BOOL;  // linked via attribute
	{attribute 'TcLinkTo' := 'TIID^Gerät 2 (EtherCAT)^Klemme 1 (EK1200)^Klemme 2 (EL3443)^L2 Status^Current Guard Warning'}
	MDP5001_341_L2_Status_Current_Guard_Warning AT%I*  : BOOL;  // linked via attribute
	{attribute 'TcLinkTo' := 'TIID^Gerät 2 (EtherCAT)^Klemme 1 (EK1200)^Klemme 2 (EL3443)^L2 Status^Current Guard Error'}
	MDP5001_341_L2_Status_Current_Guard_Error	AT%I*  : BOOL;  // linked via attribute
	{attribute 'TcLinkTo' := 'TIID^Gerät 2 (EtherCAT)^Klemme 1 (EK1200)^Klemme 2 (EL3443)^L2 Status^TxPDO Toggle'}
	MDP5001_341_L2_Status_TxPDO_Toggle			AT%I*  : BOOL;  // linked via attribute
	{attribute 'TcLinkTo' := 'TIID^Gerät 2 (EtherCAT)^Klemme 1 (EK1200)^Klemme 2 (EL3443)^L2 Basic^Voltage'}
	MDP5001_341_L2_Basic_Voltage				AT%I* : REAL;		// linked via attribute 
	{attribute 'TcLinkTo' := 'TIID^Gerät 2 (EtherCAT)^Klemme 1 (EK1200)^Klemme 2 (EL3443)^L2 Basic^Current'}
	MDP5001_341_L2_Basic_Current				AT%I* : REAL;		// linked via attribute 
	{attribute 'TcLinkTo' := 'TIID^Gerät 2 (EtherCAT)^Klemme 1 (EK1200)^Klemme 2 (EL3443)^L2 Power^Active Power'}
	MDP5001_341_L2_Power_Active_Power			AT%I* : REAL;		// linked via attribute 
	{attribute 'TcLinkTo' := 'TIID^Gerät 2 (EtherCAT)^Klemme 1 (EK1200)^Klemme 2 (EL3443)^L2 Power^Apparent Power'}
	MDP5001_341_L2_Power_Apparent_Power			AT%I* : REAL;		// linked via attribute 
	{attribute 'TcLinkTo' := 'TIID^Gerät 2 (EtherCAT)^Klemme 1 (EK1200)^Klemme 2 (EL3443)^L2 Power^Reactive Power'}
	MDP5001_341_L2_Power_Reactive_Power			AT%I* : REAL;		// linked via attribute 
	{attribute 'TcLinkTo' := 'TIID^Gerät 2 (EtherCAT)^Klemme 1 (EK1200)^Klemme 2 (EL3443)^L2 Power^Power Factor'}
	MDP5001_341_L2_Power_Power_Factor			AT%I* : REAL;		// linked via attribute 
	{attribute 'TcLinkTo' := 'TIID^Gerät 2 (EtherCAT)^Klemme 1 (EK1200)^Klemme 2 (EL3443)^L3 Status^Voltage Sign Bit'}
	MDP5001_341_L3_Status_Voltage_Sign_Bit   	AT%I*  : BOOL;  // linked via attribute 
	{attribute 'TcLinkTo' := 'TIID^Gerät 2 (EtherCAT)^Klemme 1 (EK1200)^Klemme 2 (EL3443)^L3 Status^Overvoltage'}
	MDP5001_341_L3_Status_Overvoltage			AT%I*  : BOOL;  // linked via attribute 
	{attribute 'TcLinkTo' := 'TIID^Gerät 2 (EtherCAT)^Klemme 1 (EK1200)^Klemme 2 (EL3443)^L3 Status^Overcurrent'}
	MDP5001_341_L3_Status_Overcurrent			AT%I*  : BOOL;  // linked via attribute 
	{attribute 'TcLinkTo' := 'TIID^Gerät 2 (EtherCAT)^Klemme 1 (EK1200)^Klemme 2 (EL3443)^L3 Status^Inaccurate Voltage'}	
	MDP5001_341_L3_Status_Inaccurate_Voltage	AT%I*  : BOOL;  // linked via attribute 
	{attribute 'TcLinkTo' := 'TIID^Gerät 2 (EtherCAT)^Klemme 1 (EK1200)^Klemme 2 (EL3443)^L3 Status^Inaccurate Current'}
	MDP5001_341_L3_Status_Inaccurate_Current	AT%I*  : BOOL;  // linked via attribute 	
	{attribute 'TcLinkTo' := 'TIID^Gerät 2 (EtherCAT)^Klemme 1 (EK1200)^Klemme 2 (EL3443)^L3 Status^Voltage Guard Warning'}
	MDP5001_341_L3_Status_Voltage_Guard_Warning	AT%I*  : BOOL;  // linked via attribute
	{attribute 'TcLinkTo' := 'TIID^Gerät 2 (EtherCAT)^Klemme 1 (EK1200)^Klemme 2 (EL3443)^L3 Status^Voltage Guard Error'}
	MDP5001_341_L3_Status_Voltage_Guard_Error	AT%I*  : BOOL;  // linked via attribute
	{attribute 'TcLinkTo' := 'TIID^Gerät 2 (EtherCAT)^Klemme 1 (EK1200)^Klemme 2 (EL3443)^L3 Status^Current Guard Warning'}
	MDP5001_341_L3_Status_Current_Guard_Warning AT%I*  : BOOL;  // linked via attribute
	{attribute 'TcLinkTo' := 'TIID^Gerät 2 (EtherCAT)^Klemme 1 (EK1200)^Klemme 2 (EL3443)^L3 Status^Current Guard Error'}
	MDP5001_341_L3_Status_Current_Guard_Error	AT%I*  : BOOL;  // linked via attribute
	{attribute 'TcLinkTo' := 'TIID^Gerät 2 (EtherCAT)^Klemme 1 (EK1200)^Klemme 2 (EL3443)^L3 Status^TxPDO Toggle'}
	MDP5001_341_L3_Status_TxPDO_Toggle			AT%I*  : BOOL;  // linked via attribute
	{attribute 'TcLinkTo' := 'TIID^Gerät 2 (EtherCAT)^Klemme 1 (EK1200)^Klemme 2 (EL3443)^L3 Basic^Voltage'}
	MDP5001_341_L3_Basic_Voltage				AT%I* : REAL;		// linked via attribute 
	{attribute 'TcLinkTo' := 'TIID^Gerät 2 (EtherCAT)^Klemme 1 (EK1200)^Klemme 2 (EL3443)^L3 Basic^Current'}
	MDP5001_341_L3_Basic_Current				AT%I* : REAL;		// linked via attribute 
	{attribute 'TcLinkTo' := 'TIID^Gerät 2 (EtherCAT)^Klemme 1 (EK1200)^Klemme 2 (EL3443)^L3 Power^Active Power'}
	MDP5001_341_L3_Power_Active_Power			AT%I* : REAL;		// linked via attribute 
	{attribute 'TcLinkTo' := 'TIID^Gerät 2 (EtherCAT)^Klemme 1 (EK1200)^Klemme 2 (EL3443)^L3 Power^Apparent Power'}
	MDP5001_341_L3_Power_Apparent_Power			AT%I* : REAL;		// linked via attribute 
	{attribute 'TcLinkTo' := 'TIID^Gerät 2 (EtherCAT)^Klemme 1 (EK1200)^Klemme 2 (EL3443)^L3 Power^Reactive Power'}
	MDP5001_341_L3_Power_Reactive_Power			AT%I* : REAL;		// linked via attribute 
	{attribute 'TcLinkTo' := 'TIID^Gerät 2 (EtherCAT)^Klemme 1 (EK1200)^Klemme 2 (EL3443)^L3 Power^Power Factor'}
	MDP5001_341_L3_Power_Power_Factor			AT%I* : REAL;		// linked via attribute 
	{attribute 'TcLinkTo' := 'TIID^Gerät 2 (EtherCAT)^Klemme 1 (EK1200)^Klemme 2 (EL3443)^Total Status^System State'}
	MDP5001_341_Total_Status_System_State				AT%I* : BOOL;		// linked via attribute 
	{attribute 'TcLinkTo' := 'TIID^Gerät 2 (EtherCAT)^Klemme 1 (EK1200)^Klemme 2 (EL3443)^Total Status^Grid Direction'}
	MDP5001_341_Total_Status_Grid_Direction				AT%I* : BOOL;		// linked via attribute 
	{attribute 'TcLinkTo' := 'TIID^Gerät 2 (EtherCAT)^Klemme 1 (EK1200)^Klemme 2 (EL3443)^Total Status^Frequency Guard Warning'}
	MDP5001_341_Total_Status_Frequency_Guard_Warning	AT%I* : BOOL;		// linked via attribute 
	{attribute 'TcLinkTo' := 'TIID^Gerät 2 (EtherCAT)^Klemme 1 (EK1200)^Klemme 2 (EL3443)^Total Status^Frequency Guard Error'}
	MDP5001_341_Total_Status_Frequency_Guard_Error		AT%I* : BOOL;		// linked via attribute 
	{attribute 'TcLinkTo' := 'TIID^Gerät 2 (EtherCAT)^Klemme 1 (EK1200)^Klemme 2 (EL3443)^Total Status^Neutral Current Guard Warning'}
	MDP5001_341_Total_Status_Neutral_Current_Guard_Warning	AT%I* : BOOL;		// linked via attribute 
	{attribute 'TcLinkTo' := 'TIID^Gerät 2 (EtherCAT)^Klemme 1 (EK1200)^Klemme 2 (EL3443)^Total Status^Neutral Current Guard Error'}
	MDP5001_341_Total_Status_Neutral_Current_Guard_Error	AT%I* : BOOL;		// linked via attribute 
	{attribute 'TcLinkTo' := 'TIID^Gerät 2 (EtherCAT)^Klemme 1 (EK1200)^Klemme 2 (EL3443)^Total Status^Active Power Guard Warning'}
	MDP5001_341_Total_Status_Active_Power_Guard_Warning		AT%I* : BOOL;		// linked via attribute 
	{attribute 'TcLinkTo' := 'TIID^Gerät 2 (EtherCAT)^Klemme 1 (EK1200)^Klemme 2 (EL3443)^Total Status^Active Power Guard Error'}
	MDP5001_341_Total_Status_Active_Power_Guard_Error		AT%I* : BOOL;		// linked via attribute 
	{attribute 'TcLinkTo' := 'TIID^Gerät 2 (EtherCAT)^Klemme 1 (EK1200)^Klemme 2 (EL3443)^Total Status^Apparent Power Guard Warning'}
	MDP5001_341_Total_Status_Apparent_Power_Guard_Warning	AT%I* : BOOL;		// linked via attribute 
	{attribute 'TcLinkTo' := 'TIID^Gerät 2 (EtherCAT)^Klemme 1 (EK1200)^Klemme 2 (EL3443)^Total Status^Apparent Power Guard Error'}
	MDP5001_341_Total_Status_Apparent_Power_Guard_Error		AT%I* : BOOL;		// linked via attribute 
	{attribute 'TcLinkTo' := 'TIID^Gerät 2 (EtherCAT)^Klemme 1 (EK1200)^Klemme 2 (EL3443)^Total Status^Power Quality Guard Warning'}
	MDP5001_341_Total_Status_Power_Quality_Guard_Warning	AT%I* : BOOL;		// linked via attribute 
	{attribute 'TcLinkTo' := 'TIID^Gerät 2 (EtherCAT)^Klemme 1 (EK1200)^Klemme 2 (EL3443)^Total Status^Power Quality Guard Error'}
	MDP5001_341_Total_Status_Power_Quality_Guard_Error		AT%I* : BOOL;		// linked via attribute 
	{attribute 'TcLinkTo' := 'TIID^Gerät 2 (EtherCAT)^Klemme 1 (EK1200)^Klemme 2 (EL3443)^Total Status^TxPDO State'}
	MDP5001_341_Total_Status_TxPDO_State					AT%I* : BOOL;		// linked via attribute 
	{attribute 'TcLinkTo' := 'TIID^Gerät 2 (EtherCAT)^Klemme 1 (EK1200)^Klemme 2 (EL3443)^Total Status^TxPDO Toggle'}
	MDP5001_341_Total_Status_TxPDO_Toggle					AT%I* : BOOL;		// linked via attribute 
	{attribute 'TcLinkTo' := 'TIID^Gerät 2 (EtherCAT)^Klemme 1 (EK1200)^Klemme 2 (EL3443)^Total Status^Power Quality Factor'}
	MDP5001_341_Total_Status_Power_Quality_Factor			AT%I* : REAL;		// linked via attribute 
	{attribute 'TcLinkTo' := 'TIID^Gerät 2 (EtherCAT)^Klemme 1 (EK1200)^Klemme 2 (EL3443)^Total Basic^Frequency'}
	MDP5001_341_Total_Basic_Frequency						AT%I* : REAL;		// linked via attribute 
	{attribute 'TcLinkTo' := 'TIID^Gerät 2 (EtherCAT)^Klemme 1 (EK1200)^Klemme 2 (EL3443)^Total Basic^Power Factor'}
	MDP5001_341_Total_Basic_Power_Factor					AT%I* : REAL;		// linked via attribute 
	{attribute 'TcLinkTo' := 'TIID^Gerät 2 (EtherCAT)^Klemme 1 (EK1200)^Klemme 2 (EL3443)^Total Basic^Calculated Neutral Line Current'}
	MDP5001_341_Total_Basic_Calculated_Neutral_Line_Current	AT%I* : REAL;		// linked via attribute 
	{attribute 'TcLinkTo' := 'TIID^Gerät 2 (EtherCAT)^Klemme 1 (EK1200)^Klemme 2 (EL3443)^Total Variant Value In^TxPDO Toggle'}
	MDP5001_341_Total_Variant_Value_In_TxPDO_Toggle			AT%I* : BOOL;		// linked via attribute 
	{attribute 'TcLinkTo' := 'TIID^Gerät 2 (EtherCAT)^Klemme 1 (EK1200)^Klemme 2 (EL3443)^Total Variant Value In^Index 1 REAL'}
	MDP5001_341_Total_Variant_Value_In_Index_1_REAL			AT%I* : UINT;		// linked via attribute 
	{attribute 'TcLinkTo' := 'TIID^Gerät 2 (EtherCAT)^Klemme 1 (EK1200)^Klemme 2 (EL3443)^Total Variant Value In^Value 1 REAL'}
	MDP5001_341_Total_Variant_Value_In_Value_1_REAL			AT%I* : REAL;		// linked via attribute 
	{attribute 'TcLinkTo' := 'TIID^Gerät 2 (EtherCAT)^Klemme 1 (EK1200)^Klemme 2 (EL3443)^Total Variant Value In^Index 2 REAL'}
	MDP5001_341_Total_Variant_Value_In_Index_2_REAL			AT%I* : UINT;		// linked via attribute 
	{attribute 'TcLinkTo' := 'TIID^Gerät 2 (EtherCAT)^Klemme 1 (EK1200)^Klemme 2 (EL3443)^Total Variant Value In^Value 2 REAL'}
	MDP5001_341_Total_Variant_Value_In_Value_2_REAL			AT%I* : REAL;		// linked via attribute 
	{attribute 'TcLinkTo' := 'TIID^Gerät 2 (EtherCAT)^Klemme 1 (EK1200)^Klemme 2 (EL3443)^Total Variant Value In^Index 3 REAL'}
	MDP5001_341_Total_Variant_Value_In_Index_3_REAL			AT%I* : UINT;		// linked via attribute 
	{attribute 'TcLinkTo' := 'TIID^Gerät 2 (EtherCAT)^Klemme 1 (EK1200)^Klemme 2 (EL3443)^Total Variant Value In^Value 3 REAL'}
	MDP5001_341_Total_Variant_Value_In_Value_3_REAL			AT%I* : REAL;		// linked via attribute 
	{attribute 'TcLinkTo' := 'TIID^Gerät 2 (EtherCAT)^Klemme 1 (EK1200)^Klemme 2 (EL3443)^Total Variant Value In^Index 4 ULINT'}
	MDP5001_341_Total_Variant_Value_In_Index_4_ULINT		AT%I* : UINT;		// linked via attribute 
	{attribute 'TcLinkTo' := 'TIID^Gerät 2 (EtherCAT)^Klemme 1 (EK1200)^Klemme 2 (EL3443)^Total Variant Value In^Value 4 ULINT'}
	MDP5001_341_Total_Variant_Value_In_Value_4_ULINT		AT%I* : ULINT;	// linked via attribute 
	{attribute 'TcLinkTo' := 'TIID^Gerät 2 (EtherCAT)^Klemme 1 (EK1200)^Klemme 2 (EL3443)^DPM Data^Data 1'}
	MDP5001_341_DPM_Data_Data_1								AT%I* : UDINT;	// linked via attribute 
	{attribute 'TcLinkTo' := 'TIID^Gerät 2 (EtherCAT)^Klemme 1 (EK1200)^Klemme 2 (EL3443)^DPM Data^Data 2'}
	MDP5001_341_DPM_Data_Data_2								AT%I* : UDINT;	// linked via attribute 
	{attribute 'TcLinkTo' := 'TIID^Gerät 2 (EtherCAT)^Klemme 1 (EK1200)^Klemme 2 (EL3443)^DPM Data^Data 3'}
	MDP5001_341_DPM_Data_Data_3								AT%I* : UDINT;	// linked via attribute 
	{attribute 'TcLinkTo' := 'TIID^Gerät 2 (EtherCAT)^Klemme 1 (EK1200)^Klemme 2 (EL3443)^DPM Data^Data 4'}
	MDP5001_341_DPM_Data_Data_4								AT%I* : UDINT;	// linked via attribute 
	{attribute 'TcLinkTo' := 'TIID^Gerät 2 (EtherCAT)^Klemme 1 (EK1200)^Klemme 2 (EL3443)^DPM Data^Data 5'}
	MDP5001_341_DPM_Data_Data_5								AT%I* : UDINT;	// linked via attribute 
	{attribute 'TcLinkTo' := 'TIID^Gerät 2 (EtherCAT)^Klemme 1 (EK1200)^Klemme 2 (EL3443)^DPM Data^Data 6'}
	MDP5001_341_DPM_Data_Data_6								AT%I* : UDINT;	// linked via attribute 
	{attribute 'TcLinkTo' := 'TIID^Gerät 2 (EtherCAT)^Klemme 1 (EK1200)^Klemme 2 (EL3443)^DPM Data^Data 7'}
	MDP5001_341_DPM_Data_Data_7								AT%I* : UDINT;	// linked via attribute 
	{attribute 'TcLinkTo' := 'TIID^Gerät 2 (EtherCAT)^Klemme 1 (EK1200)^Klemme 2 (EL3443)^DPM Data^Data 8'}
	MDP5001_341_DPM_Data_Data_8								AT%I* : UDINT;	// linked via attribute 
	{attribute 'TcLinkTo' := 'TIID^Gerät 2 (EtherCAT)^Klemme 1 (EK1200)^Klemme 2 (EL3443)^DPM Data^Data 9'}
	MDP5001_341_DPM_Data_Data_9								AT%I* : UDINT;	// linked via attribute 
	{attribute 'TcLinkTo' := 'TIID^Gerät 2 (EtherCAT)^Klemme 1 (EK1200)^Klemme 2 (EL3443)^DPM Data^Data 10'}
	MDP5001_341_DPM_Data_Data_10							AT%I* : UDINT;	// linked via attribute 
	{attribute 'TcLinkTo' := 'TIID^Gerät 2 (EtherCAT)^Klemme 1 (EK1200)^Klemme 2 (EL3443)^DPM Data^Data 11'}
	MDP5001_341_DPM_Data_Data_11							AT%I* : UDINT;	// linked via attribute 
	{attribute 'TcLinkTo' := 'TIID^Gerät 2 (EtherCAT)^Klemme 1 (EK1200)^Klemme 2 (EL3443)^DPM Data^Data 12'}
	MDP5001_341_DPM_Data_Data_12							AT%I* : UDINT;	// linked via attribute 
	{attribute 'TcLinkTo' := 'TIID^Gerät 2 (EtherCAT)^Klemme 1 (EK1200)^Klemme 2 (EL3443)^DPM Data^Data 13'}
	MDP5001_341_DPM_Data_Data_13							AT%I* : UDINT;	// linked via attribute 
	{attribute 'TcLinkTo' := 'TIID^Gerät 2 (EtherCAT)^Klemme 1 (EK1200)^Klemme 2 (EL3443)^DPM Data^Data 14'}
	MDP5001_341_DPM_Data_Data_14							AT%I* : UDINT;	// linked via attribute 
	{attribute 'TcLinkTo' := 'TIID^Gerät 2 (EtherCAT)^Klemme 1 (EK1200)^Klemme 2 (EL3443)^DPM Data^Data 15'}
	MDP5001_341_DPM_Data_Data_15							AT%I* : UDINT;	// linked via attribute 
	{attribute 'TcLinkTo' := 'TIID^Gerät 2 (EtherCAT)^Klemme 1 (EK1200)^Klemme 2 (EL3443)^DPM Data^Data 16'}
	MDP5001_341_DPM_Data_Data_16							AT%I* : UDINT;	// linked via attribute 
	{attribute 'TcLinkTo' := 'TIID^Gerät 2 (EtherCAT)^Klemme 1 (EK1200)^Klemme 2 (EL3443)^DPM Data^Data 17'}
	MDP5001_341_DPM_Data_Data_17							AT%I* : UDINT;	// linked via attribute 
	{attribute 'TcLinkTo' := 'TIID^Gerät 2 (EtherCAT)^Klemme 1 (EK1200)^Klemme 2 (EL3443)^DPM Data^Data 18'}
	MDP5001_341_DPM_Data_Data_18							AT%I* : UDINT;	// linked via attribute 
	{attribute 'TcLinkTo' := 'TIID^Gerät 2 (EtherCAT)^Klemme 1 (EK1200)^Klemme 2 (EL3443)^DPM Data^Data 19'}
	MDP5001_341_DPM_Data_Data_19							AT%I* : UDINT;	// linked via attribute 
	{attribute 'TcLinkTo' := 'TIID^Gerät 2 (EtherCAT)^Klemme 1 (EK1200)^Klemme 2 (EL3443)^DPM Data^Data 20'}
	MDP5001_341_DPM_Data_Data_20							AT%I* : UDINT;	// linked via attribute 
	{attribute 'TcLinkTo' := 'TIID^Gerät 2 (EtherCAT)^Klemme 1 (EK1200)^Klemme 2 (EL3443)^Total Variant Value Out^Index 1 REAL'}
	MDP5001_341_Total_Variant_Value_Out_Index_1_REAL	AT%Q* : UINT;
	{attribute 'TcLinkTo' := 'TIID^Gerät 2 (EtherCAT)^Klemme 1 (EK1200)^Klemme 2 (EL3443)^Total Variant Value Out^Index 2 REAL'}
	MDP5001_341_Total_Variant_Value_Out_Index_2_REAL	AT%Q* : UINT;
	{attribute 'TcLinkTo' := 'TIID^Gerät 2 (EtherCAT)^Klemme 1 (EK1200)^Klemme 2 (EL3443)^Total Variant Value Out^Index 3 REAL'}
	MDP5001_341_Total_Variant_Value_Out_Index_3_REAL	AT%Q* : UINT;
	{attribute 'TcLinkTo' := 'TIID^Gerät 2 (EtherCAT)^Klemme 1 (EK1200)^Klemme 2 (EL3443)^Total Variant Value Out^Index 4 ULINT'}
	MDP5001_341_Total_Variant_Value_Out_Index_4_ULINT	AT%Q* : UINT;
	{attribute 'TcLinkTo' := 'TIID^Gerät 2 (EtherCAT)^Klemme 1 (EK1200)^Klemme 2 (EL3443)^Total Interval^Reset Interval'}
	MDP5001_341_Total_Interval_Reset_Interval			AT%Q* : BOOL;
	
// IOs for EL3446
	{attribute 'TcLinkTo' := 'TIID^Gerät 2 (EtherCAT)^Klemme 1 (EK1200)^Klemme 3 (EL3446)^I1 Channel^Overcurrent'}
	MDP5001_342_I1_Channel_Overcurrent_1						AT%I*  : BOOL;
	{attribute 'TcLinkTo' := 'TIID^Gerät 2 (EtherCAT)^Klemme 1 (EK1200)^Klemme 3 (EL3446)^I1 Channel^Inaccurate Current'}
	MDP5001_342_I1_Channel_Inaccurate_Current_1				AT%I*  : BOOL;
	{attribute 'TcLinkTo' := 'TIID^Gerät 2 (EtherCAT)^Klemme 1 (EK1200)^Klemme 3 (EL3446)^I1 Channel^Current Guard Warning'}
	MDP5001_342_I1_Channel_Current_Guard_Warning_1			AT%I*  : bool;
	{attribute 'TcLinkTo' := 'TIID^Gerät 2 (EtherCAT)^Klemme 1 (EK1200)^Klemme 3 (EL3446)^I1 Channel^Current Guard Error'}
	MDP5001_342_I1_Channel_Current_Guard_Error_1				AT%I*  : bool;
	{attribute 'TcLinkTo' := 'TIID^Gerät 2 (EtherCAT)^Klemme 1 (EK1200)^Klemme 3 (EL3446)^I1 Channel^Apparent Power Guard Warning'}
	MDP5001_342_I1_Channel_Apparent_Power_Guard_Warning_1		AT%I*  : bool;
	{attribute 'TcLinkTo' := 'TIID^Gerät 2 (EtherCAT)^Klemme 1 (EK1200)^Klemme 3 (EL3446)^I1 Channel^Apparent Power Guard Error'}
	MDP5001_342_I1_Channel_Apparent_Power_Guard_Error_1		AT%I*  : bool;
	{attribute 'TcLinkTo' := 'TIID^Gerät 2 (EtherCAT)^Klemme 1 (EK1200)^Klemme 3 (EL3446)^I1 Channel^Active Power Guard Warning'}
	MDP5001_342_I1_Channel_Active_Power_Guard_Warning_1		AT%I*  : bool;
	{attribute 'TcLinkTo' := 'TIID^Gerät 2 (EtherCAT)^Klemme 1 (EK1200)^Klemme 3 (EL3446)^I1 Channel^Active Power Guard Error'}
	MDP5001_342_I1_Channel_Active_Power_Guard_Error_1			AT%I*  : bool;
	{attribute 'TcLinkTo' := 'TIID^Gerät 2 (EtherCAT)^Klemme 1 (EK1200)^Klemme 3 (EL3446)^I1 Channel^Reactive Power Guard Warning'}
	MDP5001_342_I1_Channel_Reactive_Power_Guard_Warning_1		AT%I*  : bool;
	{attribute 'TcLinkTo' := 'TIID^Gerät 2 (EtherCAT)^Klemme 1 (EK1200)^Klemme 3 (EL3446)^I1 Channel^Reactive Power Guard Error'}
	MDP5001_342_I1_Channel_Reactive_Power_Guard_Error_1		AT%I*  : bool;
	{attribute 'TcLinkTo' := 'TIID^Gerät 2 (EtherCAT)^Klemme 1 (EK1200)^Klemme 3 (EL3446)^I1 Channel^DPM Inaccurate'}
	MDP5001_342_I1_Channel_DPM_Inaccurate_1					AT%I*  : bool;
	{attribute 'TcLinkTo' := 'TIID^Gerät 2 (EtherCAT)^Klemme 1 (EK1200)^Klemme 3 (EL3446)^I1 Channel^DPM Timeout'}
	MDP5001_342_I1_Channel_DPM_Timeout_1						AT%I*  : bool;
	{attribute 'TcLinkTo' := 'TIID^Gerät 2 (EtherCAT)^Klemme 1 (EK1200)^Klemme 3 (EL3446)^I1 Channel^TxPDO Toggle'}
	MDP5001_342_I1_Channel_TxPDO_Toggle_1						AT%I*  : bool;
	{attribute 'TcLinkTo' := 'TIID^Gerät 2 (EtherCAT)^Klemme 1 (EK1200)^Klemme 3 (EL3446)^I1 Channel^Current'}
	MDP5001_342_I1_Channel_Current_1							AT%I*  : REAL;
	{attribute 'TcLinkTo' := 'TIID^Gerät 2 (EtherCAT)^Klemme 1 (EK1200)^Klemme 3 (EL3446)^I1 Channel^Active Power'}
	MDP5001_342_I1_Channel_Active_Power_1						AT%I*  : REAL;
	{attribute 'TcLinkTo' := 'TIID^Gerät 2 (EtherCAT)^Klemme 1 (EK1200)^Klemme 3 (EL3446)^I1 Channel^Apparent Power'}
	MDP5001_342_I1_Channel_Apparent_Power_1					AT%I*  : REAL;
	{attribute 'TcLinkTo' := 'TIID^Gerät 2 (EtherCAT)^Klemme 1 (EK1200)^Klemme 3 (EL3446)^I1 Channel^Reactive Power Fundamental'}
	MDP5001_342_I1_Channel_Reactive_Power_Fundamental_1		AT%I*  : REAL;
	{attribute 'TcLinkTo' := 'TIID^Gerät 2 (EtherCAT)^Klemme 1 (EK1200)^Klemme 3 (EL3446)^I1 Channel^Active Energy'}
	MDP5001_342_I1_Channel_Active_Energy_1					AT%I*  : DINT;
	{attribute 'TcLinkTo' := 'TIID^Gerät 2 (EtherCAT)^Klemme 1 (EK1200)^Klemme 3 (EL3446)^I2 Channel^Overcurrent'}
	MDP5001_342_I2_Channel_Overcurrent_1						AT%I*  : BOOL;
	{attribute 'TcLinkTo' := 'TIID^Gerät 2 (EtherCAT)^Klemme 1 (EK1200)^Klemme 3 (EL3446)^I2 Channel^Inaccurate Current'}
	MDP5001_342_I2_Channel_Inaccurate_Current_1				AT%I*  : BOOL;
	{attribute 'TcLinkTo' := 'TIID^Gerät 2 (EtherCAT)^Klemme 1 (EK1200)^Klemme 3 (EL3446)^I2 Channel^Current Guard Warning'}
	MDP5001_342_I2_Channel_Current_Guard_Warning_1			AT%I*  : bool;
	{attribute 'TcLinkTo' := 'TIID^Gerät 2 (EtherCAT)^Klemme 1 (EK1200)^Klemme 3 (EL3446)^I2 Channel^Current Guard Error'}
	MDP5001_342_I2_Channel_Current_Guard_Error_1				AT%I*  : bool;
	{attribute 'TcLinkTo' := 'TIID^Gerät 2 (EtherCAT)^Klemme 1 (EK1200)^Klemme 3 (EL3446)^I2 Channel^Apparent Power Guard Warning'}
	MDP5001_342_I2_Channel_Apparent_Power_Guard_Warning_1		AT%I*  : bool;
	{attribute 'TcLinkTo' := 'TIID^Gerät 2 (EtherCAT)^Klemme 1 (EK1200)^Klemme 3 (EL3446)^I2 Channel^Apparent Power Guard Error'}
	MDP5001_342_I2_Channel_Apparent_Power_Guard_Error_1		AT%I*  : bool;
	{attribute 'TcLinkTo' := 'TIID^Gerät 2 (EtherCAT)^Klemme 1 (EK1200)^Klemme 3 (EL3446)^I2 Channel^Active Power Guard Warning'}
	MDP5001_342_I2_Channel_Active_Power_Guard_Warning_1		AT%I*  : bool;
	{attribute 'TcLinkTo' := 'TIID^Gerät 2 (EtherCAT)^Klemme 1 (EK1200)^Klemme 3 (EL3446)^I2 Channel^Active Power Guard Error'}
	MDP5001_342_I2_Channel_Active_Power_Guard_Error_1			AT%I*  : bool;
	{attribute 'TcLinkTo' := 'TIID^Gerät 2 (EtherCAT)^Klemme 1 (EK1200)^Klemme 3 (EL3446)^I2 Channel^Reactive Power Guard Warning'}
	MDP5001_342_I2_Channel_Reactive_Power_Guard_Warning_1		AT%I*  : bool;
	{attribute 'TcLinkTo' := 'TIID^Gerät 2 (EtherCAT)^Klemme 1 (EK1200)^Klemme 3 (EL3446)^I2 Channel^Reactive Power Guard Error'}
	MDP5001_342_I2_Channel_Reactive_Power_Guard_Error_1		AT%I*  : bool;
	{attribute 'TcLinkTo' := 'TIID^Gerät 2 (EtherCAT)^Klemme 1 (EK1200)^Klemme 3 (EL3446)^I2 Channel^DPM Inaccurate'}
	MDP5001_342_I2_Channel_DPM_Inaccurate_1					AT%I*  : bool;
	{attribute 'TcLinkTo' := 'TIID^Gerät 2 (EtherCAT)^Klemme 1 (EK1200)^Klemme 3 (EL3446)^I2 Channel^DPM Timeout'}
	MDP5001_342_I2_Channel_DPM_Timeout_1						AT%I*  : bool;
	{attribute 'TcLinkTo' := 'TIID^Gerät 2 (EtherCAT)^Klemme 1 (EK1200)^Klemme 3 (EL3446)^I2 Channel^TxPDO Toggle'}
	MDP5001_342_I2_Channel_TxPDO_Toggle_1						AT%I*  : bool;
	{attribute 'TcLinkTo' := 'TIID^Gerät 2 (EtherCAT)^Klemme 1 (EK1200)^Klemme 3 (EL3446)^I2 Channel^Current'}
	MDP5001_342_I2_Channel_Current_1							AT%I*  : REAL;
	{attribute 'TcLinkTo' := 'TIID^Gerät 2 (EtherCAT)^Klemme 1 (EK1200)^Klemme 3 (EL3446)^I2 Channel^Active Power'}
	MDP5001_342_I2_Channel_Active_Power_1						AT%I*  : REAL;
	{attribute 'TcLinkTo' := 'TIID^Gerät 2 (EtherCAT)^Klemme 1 (EK1200)^Klemme 3 (EL3446)^I2 Channel^Apparent Power'}
	MDP5001_342_I2_Channel_Apparent_Power_1					AT%I*  : REAL;
	{attribute 'TcLinkTo' := 'TIID^Gerät 2 (EtherCAT)^Klemme 1 (EK1200)^Klemme 3 (EL3446)^I2 Channel^Reactive Power Fundamental'}
	MDP5001_342_I2_Channel_Reactive_Power_Fundamental_1		AT%I*  : REAL;
	{attribute 'TcLinkTo' := 'TIID^Gerät 2 (EtherCAT)^Klemme 1 (EK1200)^Klemme 3 (EL3446)^I2 Channel^Active Energy'}
	MDP5001_342_I2_Channel_Active_Energy_1					AT%I*  : DINT;
	{attribute 'TcLinkTo' := 'TIID^Gerät 2 (EtherCAT)^Klemme 1 (EK1200)^Klemme 3 (EL3446)^I3 Channel^Overcurrent'}
	MDP5001_342_I3_Channel_Overcurrent_1						AT%I*  : BOOL;
	{attribute 'TcLinkTo' := 'TIID^Gerät 2 (EtherCAT)^Klemme 1 (EK1200)^Klemme 3 (EL3446)^I3 Channel^Inaccurate Current'}
	MDP5001_342_I3_Channel_Inaccurate_Current_1				AT%I*  : BOOL;
	{attribute 'TcLinkTo' := 'TIID^Gerät 2 (EtherCAT)^Klemme 1 (EK1200)^Klemme 3 (EL3446)^I3 Channel^Current Guard Warning'}
	MDP5001_342_I3_Channel_Current_Guard_Warning_1			AT%I*  : bool;
	{attribute 'TcLinkTo' := 'TIID^Gerät 2 (EtherCAT)^Klemme 1 (EK1200)^Klemme 3 (EL3446)^I3 Channel^Current Guard Error'}
	MDP5001_342_I3_Channel_Current_Guard_Error_1				AT%I*  : bool;
	{attribute 'TcLinkTo' := 'TIID^Gerät 2 (EtherCAT)^Klemme 1 (EK1200)^Klemme 3 (EL3446)^I3 Channel^Apparent Power Guard Warning'}
	MDP5001_342_I3_Channel_Apparent_Power_Guard_Warning_1		AT%I*  : bool;
	{attribute 'TcLinkTo' := 'TIID^Gerät 2 (EtherCAT)^Klemme 1 (EK1200)^Klemme 3 (EL3446)^I3 Channel^Apparent Power Guard Error'}
	MDP5001_342_I3_Channel_Apparent_Power_Guard_Error_1		AT%I*  : bool;
	{attribute 'TcLinkTo' := 'TIID^Gerät 2 (EtherCAT)^Klemme 1 (EK1200)^Klemme 3 (EL3446)^I3 Channel^Active Power Guard Warning'}
	MDP5001_342_I3_Channel_Active_Power_Guard_Warning_1		AT%I*  : bool;
	{attribute 'TcLinkTo' := 'TIID^Gerät 2 (EtherCAT)^Klemme 1 (EK1200)^Klemme 3 (EL3446)^I3 Channel^Active Power Guard Error'}
	MDP5001_342_I3_Channel_Active_Power_Guard_Error_1		AT%I*  : bool;
	{attribute 'TcLinkTo' := 'TIID^Gerät 2 (EtherCAT)^Klemme 1 (EK1200)^Klemme 3 (EL3446)^I3 Channel^Reactive Power Guard Warning'}
	MDP5001_342_I3_Channel_Reactive_Power_Guard_Warning_1		AT%I*  : bool;
	{attribute 'TcLinkTo' := 'TIID^Gerät 2 (EtherCAT)^Klemme 1 (EK1200)^Klemme 3 (EL3446)^I3 Channel^Reactive Power Guard Error'}
	MDP5001_342_I3_Channel_Reactive_Power_Guard_Error_1		AT%I*  : bool;
	{attribute 'TcLinkTo' := 'TIID^Gerät 2 (EtherCAT)^Klemme 1 (EK1200)^Klemme 3 (EL3446)^I3 Channel^DPM Inaccurate'}
	MDP5001_342_I3_Channel_DPM_Inaccurate_1					AT%I*  : bool;
	{attribute 'TcLinkTo' := 'TIID^Gerät 2 (EtherCAT)^Klemme 1 (EK1200)^Klemme 3 (EL3446)^I3 Channel^DPM Timeout'}
	MDP5001_342_I3_Channel_DPM_Timeout_1						AT%I*  : bool;
	{attribute 'TcLinkTo' := 'TIID^Gerät 2 (EtherCAT)^Klemme 1 (EK1200)^Klemme 3 (EL3446)^I3 Channel^TxPDO Toggle'}
	MDP5001_342_I3_Channel_TxPDO_Toggle_1						AT%I*  : bool;
	{attribute 'TcLinkTo' := 'TIID^Gerät 2 (EtherCAT)^Klemme 1 (EK1200)^Klemme 3 (EL3446)^I3 Channel^Current'}
	MDP5001_342_I3_Channel_Current_1							AT%I*  : REAL;
	{attribute 'TcLinkTo' := 'TIID^Gerät 2 (EtherCAT)^Klemme 1 (EK1200)^Klemme 3 (EL3446)^I3 Channel^Active Power'}
	MDP5001_342_I3_Channel_Active_Power_1						AT%I*  : REAL;
	{attribute 'TcLinkTo' := 'TIID^Gerät 2 (EtherCAT)^Klemme 1 (EK1200)^Klemme 3 (EL3446)^I3 Channel^Apparent Power'}
	MDP5001_342_I3_Channel_Apparent_Power_1					AT%I*  : REAL;
	{attribute 'TcLinkTo' := 'TIID^Gerät 2 (EtherCAT)^Klemme 1 (EK1200)^Klemme 3 (EL3446)^I3 Channel^Reactive Power Fundamental'}
	MDP5001_342_I3_Channel_Reactive_Power_Fundamental_1		AT%I*  : REAL;
	{attribute 'TcLinkTo' := 'TIID^Gerät 2 (EtherCAT)^Klemme 1 (EK1200)^Klemme 3 (EL3446)^I3 Channel^Active Energy'}
	MDP5001_342_I3_Channel_Active_Energy_1					AT%I*  : DINT;	
	{attribute 'TcLinkTo' := 'TIID^Gerät 2 (EtherCAT)^Klemme 1 (EK1200)^Klemme 3 (EL3446)^I4 Channel^Overcurrent'}
	MDP5001_342_I4_Channel_Overcurrent_1						AT%I*  : BOOL;
	{attribute 'TcLinkTo' := 'TIID^Gerät 2 (EtherCAT)^Klemme 1 (EK1200)^Klemme 3 (EL3446)^I4 Channel^Inaccurate Current'}
	MDP5001_342_I4_Channel_Inaccurate_Current_1				AT%I*  : BOOL;
	{attribute 'TcLinkTo' := 'TIID^Gerät 2 (EtherCAT)^Klemme 1 (EK1200)^Klemme 3 (EL3446)^I4 Channel^Current Guard Warning'}
	MDP5001_342_I4_Channel_Current_Guard_Warning_1			AT%I*  : bool;
	{attribute 'TcLinkTo' := 'TIID^Gerät 2 (EtherCAT)^Klemme 1 (EK1200)^Klemme 3 (EL3446)^I4 Channel^Current Guard Error'}
	MDP5001_342_I4_Channel_Current_Guard_Error_1				AT%I*  : bool;
	{attribute 'TcLinkTo' := 'TIID^Gerät 2 (EtherCAT)^Klemme 1 (EK1200)^Klemme 3 (EL3446)^I4 Channel^Apparent Power Guard Warning'}
	MDP5001_342_I4_Channel_Apparent_Power_Guard_Warning_1		AT%I*  : bool;
	{attribute 'TcLinkTo' := 'TIID^Gerät 2 (EtherCAT)^Klemme 1 (EK1200)^Klemme 3 (EL3446)^I4 Channel^Apparent Power Guard Error'}
	MDP5001_342_I4_Channel_Apparent_Power_Guard_Error_1		AT%I*  : bool;
	{attribute 'TcLinkTo' := 'TIID^Gerät 2 (EtherCAT)^Klemme 1 (EK1200)^Klemme 3 (EL3446)^I4 Channel^Active Power Guard Warning'}
	MDP5001_342_I4_Channel_Active_Power_Guard_Warning_1		AT%I*  : bool;
	{attribute 'TcLinkTo' := 'TIID^Gerät 2 (EtherCAT)^Klemme 1 (EK1200)^Klemme 3 (EL3446)^I4 Channel^Active Power Guard Error'}
	MDP5001_342_I4_Channel_Active_Power_Guard_Error_1			AT%I*  : bool;
	{attribute 'TcLinkTo' := 'TIID^Gerät 2 (EtherCAT)^Klemme 1 (EK1200)^Klemme 3 (EL3446)^I4 Channel^Reactive Power Guard Warning'}
	MDP5001_342_I4_Channel_Reactive_Power_Guard_Warning_1		AT%I*  : bool;
	{attribute 'TcLinkTo' := 'TIID^Gerät 2 (EtherCAT)^Klemme 1 (EK1200)^Klemme 3 (EL3446)^I4 Channel^Reactive Power Guard Error'}
	MDP5001_342_I4_Channel_Reactive_Power_Guard_Error_1		AT%I*  : bool;
	{attribute 'TcLinkTo' := 'TIID^Gerät 2 (EtherCAT)^Klemme 1 (EK1200)^Klemme 3 (EL3446)^I4 Channel^DPM Inaccurate'}
	MDP5001_342_I4_Channel_DPM_Inaccurate_1					AT%I*  : bool;
	{attribute 'TcLinkTo' := 'TIID^Gerät 2 (EtherCAT)^Klemme 1 (EK1200)^Klemme 3 (EL3446)^I4 Channel^DPM Timeout'}
	MDP5001_342_I4_Channel_DPM_Timeout_1						AT%I*  : bool;
	{attribute 'TcLinkTo' := 'TIID^Gerät 2 (EtherCAT)^Klemme 1 (EK1200)^Klemme 3 (EL3446)^I4 Channel^TxPDO Toggle'}
	MDP5001_342_I4_Channel_TxPDO_Toggle_1						AT%I*  : bool;
	{attribute 'TcLinkTo' := 'TIID^Gerät 2 (EtherCAT)^Klemme 1 (EK1200)^Klemme 3 (EL3446)^I4 Channel^Current'}
	MDP5001_342_I4_Channel_Current_1							AT%I*  : REAL;
	{attribute 'TcLinkTo' := 'TIID^Gerät 2 (EtherCAT)^Klemme 1 (EK1200)^Klemme 3 (EL3446)^I4 Channel^Active Power'}
	MDP5001_342_I4_Channel_Active_Power_1						AT%I*  : REAL;
	{attribute 'TcLinkTo' := 'TIID^Gerät 2 (EtherCAT)^Klemme 1 (EK1200)^Klemme 3 (EL3446)^I4 Channel^Apparent Power'}
	MDP5001_342_I4_Channel_Apparent_Power_1					AT%I*  : REAL;
	{attribute 'TcLinkTo' := 'TIID^Gerät 2 (EtherCAT)^Klemme 1 (EK1200)^Klemme 3 (EL3446)^I4 Channel^Reactive Power Fundamental'}
	MDP5001_342_I4_Channel_Reactive_Power_Fundamental_1		AT%I*  : REAL;
	{attribute 'TcLinkTo' := 'TIID^Gerät 2 (EtherCAT)^Klemme 1 (EK1200)^Klemme 3 (EL3446)^I4 Channel^Active Energy'}
	MDP5001_342_I4_Channel_Active_Energy_1					AT%I*  : DINT;
	{attribute 'TcLinkTo' := 'TIID^Gerät 2 (EtherCAT)^Klemme 1 (EK1200)^Klemme 3 (EL3446)^I5 Channel^Overcurrent'}
	MDP5001_342_I5_Channel_Overcurrent_1						AT%I*  : BOOL;
	{attribute 'TcLinkTo' := 'TIID^Gerät 2 (EtherCAT)^Klemme 1 (EK1200)^Klemme 3 (EL3446)^I5 Channel^Inaccurate Current'}
	MDP5001_342_I5_Channel_Inaccurate_Current_1				AT%I*  : BOOL;
	{attribute 'TcLinkTo' := 'TIID^Gerät 2 (EtherCAT)^Klemme 1 (EK1200)^Klemme 3 (EL3446)^I5 Channel^Current Guard Warning'}
	MDP5001_342_I5_Channel_Current_Guard_Warning_1			AT%I*  : bool;
	{attribute 'TcLinkTo' := 'TIID^Gerät 2 (EtherCAT)^Klemme 1 (EK1200)^Klemme 3 (EL3446)^I5 Channel^Current Guard Error'}
	MDP5001_342_I5_Channel_Current_Guard_Error_1				AT%I*  : bool;
	{attribute 'TcLinkTo' := 'TIID^Gerät 2 (EtherCAT)^Klemme 1 (EK1200)^Klemme 3 (EL3446)^I5 Channel^Apparent Power Guard Warning'}
	MDP5001_342_I5_Channel_Apparent_Power_Guard_Warning_1		AT%I*  : bool;
	{attribute 'TcLinkTo' := 'TIID^Gerät 2 (EtherCAT)^Klemme 1 (EK1200)^Klemme 3 (EL3446)^I5 Channel^Apparent Power Guard Error'}
	MDP5001_342_I5_Channel_Apparent_Power_Guard_Error_1		AT%I*  : bool;
	{attribute 'TcLinkTo' := 'TIID^Gerät 2 (EtherCAT)^Klemme 1 (EK1200)^Klemme 3 (EL3446)^I5 Channel^Active Power Guard Warning'}
	MDP5001_342_I5_Channel_Active_Power_Guard_Warning_1		AT%I*  : bool;
	{attribute 'TcLinkTo' := 'TIID^Gerät 2 (EtherCAT)^Klemme 1 (EK1200)^Klemme 3 (EL3446)^I5 Channel^Active Power Guard Error'}
	MDP5001_342_I5_Channel_Active_Power_Guard_Error_1			AT%I*  : bool;
	{attribute 'TcLinkTo' := 'TIID^Gerät 2 (EtherCAT)^Klemme 1 (EK1200)^Klemme 3 (EL3446)^I5 Channel^Reactive Power Guard Warning'}
	MDP5001_342_I5_Channel_Reactive_Power_Guard_Warning_1		AT%I*  : bool;
	{attribute 'TcLinkTo' := 'TIID^Gerät 2 (EtherCAT)^Klemme 1 (EK1200)^Klemme 3 (EL3446)^I5 Channel^Reactive Power Guard Error'}
	MDP5001_342_I5_Channel_Reactive_Power_Guard_Error_1		AT%I*  : bool;
	{attribute 'TcLinkTo' := 'TIID^Gerät 2 (EtherCAT)^Klemme 1 (EK1200)^Klemme 3 (EL3446)^I5 Channel^DPM Inaccurate'}
	MDP5001_342_I5_Channel_DPM_Inaccurate_1					AT%I*  : bool;
	{attribute 'TcLinkTo' := 'TIID^Gerät 2 (EtherCAT)^Klemme 1 (EK1200)^Klemme 3 (EL3446)^I5 Channel^DPM Timeout'}
	MDP5001_342_I5_Channel_DPM_Timeout_1						AT%I*  : bool;
	{attribute 'TcLinkTo' := 'TIID^Gerät 2 (EtherCAT)^Klemme 1 (EK1200)^Klemme 3 (EL3446)^I5 Channel^TxPDO Toggle'}
	MDP5001_342_I5_Channel_TxPDO_Toggle_1						AT%I*  : bool;
	{attribute 'TcLinkTo' := 'TIID^Gerät 2 (EtherCAT)^Klemme 1 (EK1200)^Klemme 3 (EL3446)^I5 Channel^Current'}
	MDP5001_342_I5_Channel_Current_1							AT%I*  : REAL;
	{attribute 'TcLinkTo' := 'TIID^Gerät 2 (EtherCAT)^Klemme 1 (EK1200)^Klemme 3 (EL3446)^I5 Channel^Active Power'}
	MDP5001_342_I5_Channel_Active_Power_1						AT%I*  : REAL;
	{attribute 'TcLinkTo' := 'TIID^Gerät 2 (EtherCAT)^Klemme 1 (EK1200)^Klemme 3 (EL3446)^I5 Channel^Apparent Power'}
	MDP5001_342_I5_Channel_Apparent_Power_1					AT%I*  : REAL;
	{attribute 'TcLinkTo' := 'TIID^Gerät 2 (EtherCAT)^Klemme 1 (EK1200)^Klemme 3 (EL3446)^I5 Channel^Reactive Power Fundamental'}
	MDP5001_342_I5_Channel_Reactive_Power_Fundamental_1		AT%I*  : REAL;
	{attribute 'TcLinkTo' := 'TIID^Gerät 2 (EtherCAT)^Klemme 1 (EK1200)^Klemme 3 (EL3446)^I5 Channel^Active Energy'}
	MDP5001_342_I5_Channel_Active_Energy_1					AT%I*  : DINT;
	{attribute 'TcLinkTo' := 'TIID^Gerät 2 (EtherCAT)^Klemme 1 (EK1200)^Klemme 3 (EL3446)^I6 Channel^Overcurrent'}
	MDP5001_342_I6_Channel_Overcurrent_1						AT%I*  : BOOL;
	{attribute 'TcLinkTo' := 'TIID^Gerät 2 (EtherCAT)^Klemme 1 (EK1200)^Klemme 3 (EL3446)^I6 Channel^Inaccurate Current'}
	MDP5001_342_I6_Channel_Inaccurate_Current_1				AT%I*  : BOOL;
	{attribute 'TcLinkTo' := 'TIID^Gerät 2 (EtherCAT)^Klemme 1 (EK1200)^Klemme 3 (EL3446)^I6 Channel^Current Guard Warning'}
	MDP5001_342_I6_Channel_Current_Guard_Warning_1			AT%I*  : bool;
	{attribute 'TcLinkTo' := 'TIID^Gerät 2 (EtherCAT)^Klemme 1 (EK1200)^Klemme 3 (EL3446)^I6 Channel^Current Guard Error'}
	MDP5001_342_I6_Channel_Current_Guard_Error_1				AT%I*  : bool;
	{attribute 'TcLinkTo' := 'TIID^Gerät 2 (EtherCAT)^Klemme 1 (EK1200)^Klemme 3 (EL3446)^I6 Channel^Apparent Power Guard Warning'}
	MDP5001_342_I6_Channel_Apparent_Power_Guard_Warning_1		AT%I*  : bool;
	{attribute 'TcLinkTo' := 'TIID^Gerät 2 (EtherCAT)^Klemme 1 (EK1200)^Klemme 3 (EL3446)^I6 Channel^Apparent Power Guard Error'}
	MDP5001_342_I6_Channel_Apparent_Power_Guard_Error_1		AT%I*  : bool;
	{attribute 'TcLinkTo' := 'TIID^Gerät 2 (EtherCAT)^Klemme 1 (EK1200)^Klemme 3 (EL3446)^I6 Channel^Active Power Guard Warning'}
	MDP5001_342_I6_Channel_Active_Power_Guard_Warning_1		AT%I*  : bool;
	{attribute 'TcLinkTo' := 'TIID^Gerät 2 (EtherCAT)^Klemme 1 (EK1200)^Klemme 3 (EL3446)^I6 Channel^Active Power Guard Error'}
	MDP5001_342_I6_Channel_Active_Power_Guard_Error_1			AT%I*  : bool;
	{attribute 'TcLinkTo' := 'TIID^Gerät 2 (EtherCAT)^Klemme 1 (EK1200)^Klemme 3 (EL3446)^I6 Channel^Reactive Power Guard Warning'}
	MDP5001_342_I6_Channel_Reactive_Power_Guard_Warning_1		AT%I*  : bool;
	{attribute 'TcLinkTo' := 'TIID^Gerät 2 (EtherCAT)^Klemme 1 (EK1200)^Klemme 3 (EL3446)^I6 Channel^Reactive Power Guard Error'}
	MDP5001_342_I6_Channel_Reactive_Power_Guard_Error_1		AT%I*  : bool;
	{attribute 'TcLinkTo' := 'TIID^Gerät 2 (EtherCAT)^Klemme 1 (EK1200)^Klemme 3 (EL3446)^I6 Channel^DPM Inaccurate'}
	MDP5001_342_I6_Channel_DPM_Inaccurate_1					AT%I*  : bool;
	{attribute 'TcLinkTo' := 'TIID^Gerät 2 (EtherCAT)^Klemme 1 (EK1200)^Klemme 3 (EL3446)^I6 Channel^DPM Timeout'}
	MDP5001_342_I6_Channel_DPM_Timeout_1						AT%I*  : bool;
	{attribute 'TcLinkTo' := 'TIID^Gerät 2 (EtherCAT)^Klemme 1 (EK1200)^Klemme 3 (EL3446)^I6 Channel^TxPDO Toggle'}
	MDP5001_342_I6_Channel_TxPDO_Toggle_1						AT%I*  : bool;
	{attribute 'TcLinkTo' := 'TIID^Gerät 2 (EtherCAT)^Klemme 1 (EK1200)^Klemme 3 (EL3446)^I6 Channel^Current'}
	MDP5001_342_I6_Channel_Current_1							AT%I*  : REAL;
	{attribute 'TcLinkTo' := 'TIID^Gerät 2 (EtherCAT)^Klemme 1 (EK1200)^Klemme 3 (EL3446)^I6 Channel^Active Power'}
	MDP5001_342_I6_Channel_Active_Power_1						AT%I*  : REAL;
	{attribute 'TcLinkTo' := 'TIID^Gerät 2 (EtherCAT)^Klemme 1 (EK1200)^Klemme 3 (EL3446)^I6 Channel^Apparent Power'}
	MDP5001_342_I6_Channel_Apparent_Power_1					AT%I*  : REAL;
	{attribute 'TcLinkTo' := 'TIID^Gerät 2 (EtherCAT)^Klemme 1 (EK1200)^Klemme 3 (EL3446)^I6 Channel^Reactive Power Fundamental'}
	MDP5001_342_I6_Channel_Reactive_Power_Fundamental_1		AT%I*  : REAL;
	{attribute 'TcLinkTo' := 'TIID^Gerät 2 (EtherCAT)^Klemme 1 (EK1200)^Klemme 3 (EL3446)^I6 Channel^Active Energy'}
	MDP5001_342_I6_Channel_Active_Energy_1					AT%I*  : DINT;	
	
	{attribute 'TcLinkTo' := 'TIID^Gerät 2 (EtherCAT)^Klemme 1 (EK1200)^Klemme 3 (EL3446)^DPM Variant Value In^TxPDO Toggle'}
	MDP5001_342_DPM_Variant_Value_In_TxPDO_Toggle_1			AT%I*  : BOOL;
	{attribute 'TcLinkTo' := 'TIID^Gerät 2 (EtherCAT)^Klemme 1 (EK1200)^Klemme 3 (EL3446)^DPM Variant Value In^Index 1 REAL'}
	MDP5001_342_DPM_Variant_Value_In_Index_1_REAL_1			AT%I*  : UINT;
	{attribute 'TcLinkTo' := 'TIID^Gerät 2 (EtherCAT)^Klemme 1 (EK1200)^Klemme 3 (EL3446)^DPM Variant Value In^Value 1 REAL'}
	MDP5001_342_DPM_Variant_Value_In_Value_1_REAL_1			AT%I*  : REAL;
	{attribute 'TcLinkTo' := 'TIID^Gerät 2 (EtherCAT)^Klemme 1 (EK1200)^Klemme 3 (EL3446)^DPM Variant Value In^Index 2 REAL'}
	MDP5001_342_DPM_Variant_Value_In_Index_2_REAL_1			AT%I*  : UINT;
	{attribute 'TcLinkTo' := 'TIID^Gerät 2 (EtherCAT)^Klemme 1 (EK1200)^Klemme 3 (EL3446)^DPM Variant Value In^Value 2 REAL'}
	MDP5001_342_DPM_Variant_Value_In_Value_2_REAL_1			AT%I*  : REAL;
	{attribute 'TcLinkTo' := 'TIID^Gerät 2 (EtherCAT)^Klemme 1 (EK1200)^Klemme 3 (EL3446)^DPM Variant Value In^Index 3 REAL'}
	MDP5001_342_DPM_Variant_Value_In_Index_3_REAL_1			AT%I*  : UINT;
	{attribute 'TcLinkTo' := 'TIID^Gerät 2 (EtherCAT)^Klemme 1 (EK1200)^Klemme 3 (EL3446)^DPM Variant Value In^Value 3 REAL'}
	MDP5001_342_DPM_Variant_Value_In_Value_3_REAL_1			AT%I*  : REAL;
	{attribute 'TcLinkTo' := 'TIID^Gerät 2 (EtherCAT)^Klemme 1 (EK1200)^Klemme 3 (EL3446)^DPM Variant Value In^Index 4 ULINT'}
	MDP5001_342_DPM_Variant_Value_In_Index_4_ULINT_1			AT%I*  : UINT;
	{attribute 'TcLinkTo' := 'TIID^Gerät 2 (EtherCAT)^Klemme 1 (EK1200)^Klemme 3 (EL3446)^DPM Variant Value In^Value 4 ULINT'}
	MDP5001_342_DPM_Variant_Value_In_Value_4_ULINT_1			AT%I*  : ULINT;

	{attribute 'TcLinkTo' := 'TIID^Gerät 2 (EtherCAT)^Klemme 1 (EK1200)^Klemme 3 (EL3446)^DPM Variant Value Out^Index 1 REAL'}
	MDP5001_342_DPM_Variant_Value_Out_Index_1_REAL_1	AT%Q* : UINT;
	{attribute 'TcLinkTo' := 'TIID^Gerät 2 (EtherCAT)^Klemme 1 (EK1200)^Klemme 3 (EL3446)^DPM Variant Value Out^Index 2 REAL'}
	MDP5001_342_DPM_Variant_Value_Out_Index_2_REAL_1	AT%Q* : UINT;
	{attribute 'TcLinkTo' := 'TIID^Gerät 2 (EtherCAT)^Klemme 1 (EK1200)^Klemme 3 (EL3446)^DPM Variant Value Out^Index 3 REAL'}
	MDP5001_342_DPM_Variant_Value_Out_Index_3_REAL_1	AT%Q* : UINT;
	{attribute 'TcLinkTo' := 'TIID^Gerät 2 (EtherCAT)^Klemme 1 (EK1200)^Klemme 3 (EL3446)^DPM Variant Value Out^Index 4 ULINT'}
	MDP5001_342_DPM_Variant_Value_Out_Index_4_ULINT_1	AT%Q* : UINT;
	{attribute 'TcLinkTo' := 'TIID^Gerät 2 (EtherCAT)^Klemme 1 (EK1200)^Klemme 3 (EL3446)^DPM Data^Data 1'}
	MDP5001_342_DPM_Data_Data_1_1						AT%Q* : UDINT;
	{attribute 'TcLinkTo' := 'TIID^Gerät 2 (EtherCAT)^Klemme 1 (EK1200)^Klemme 3 (EL3446)^DPM Data^Data 2'}
	MDP5001_342_DPM_Data_Data_2_1						AT%Q* : UDINT;
	{attribute 'TcLinkTo' := 'TIID^Gerät 2 (EtherCAT)^Klemme 1 (EK1200)^Klemme 3 (EL3446)^DPM Data^Data 3'}
	MDP5001_342_DPM_Data_Data_3_1						AT%Q* : UDINT;
	{attribute 'TcLinkTo' := 'TIID^Gerät 2 (EtherCAT)^Klemme 1 (EK1200)^Klemme 3 (EL3446)^DPM Data^Data 4'}
	MDP5001_342_DPM_Data_Data_4_1						AT%Q* : UDINT;
	{attribute 'TcLinkTo' := 'TIID^Gerät 2 (EtherCAT)^Klemme 1 (EK1200)^Klemme 3 (EL3446)^DPM Data^Data 5'}
	MDP5001_342_DPM_Data_Data_5_1						AT%Q* : UDINT;
	{attribute 'TcLinkTo' := 'TIID^Gerät 2 (EtherCAT)^Klemme 1 (EK1200)^Klemme 3 (EL3446)^DPM Data^Data 6'}
	MDP5001_342_DPM_Data_Data_6_1						AT%Q* : UDINT;
	{attribute 'TcLinkTo' := 'TIID^Gerät 2 (EtherCAT)^Klemme 1 (EK1200)^Klemme 3 (EL3446)^DPM Data^Data 7'}
	MDP5001_342_DPM_Data_Data_7_1						AT%Q* : UDINT;
	{attribute 'TcLinkTo' := 'TIID^Gerät 2 (EtherCAT)^Klemme 1 (EK1200)^Klemme 3 (EL3446)^DPM Data^Data 8'}
	MDP5001_342_DPM_Data_Data_8_1						AT%Q* : UDINT;
	{attribute 'TcLinkTo' := 'TIID^Gerät 2 (EtherCAT)^Klemme 1 (EK1200)^Klemme 3 (EL3446)^DPM Data^Data 9'}
	MDP5001_342_DPM_Data_Data_9_1						AT%Q* : UDINT;
	{attribute 'TcLinkTo' := 'TIID^Gerät 2 (EtherCAT)^Klemme 1 (EK1200)^Klemme 3 (EL3446)^DPM Data^Data 10'}
	MDP5001_342_DPM_Data_Data_10_1					AT%Q* : UDINT;
	{attribute 'TcLinkTo' := 'TIID^Gerät 2 (EtherCAT)^Klemme 1 (EK1200)^Klemme 3 (EL3446)^DPM Data^Data 11'}
	MDP5001_342_DPM_Data_Data_11_1					AT%Q* : UDINT;
	{attribute 'TcLinkTo' := 'TIID^Gerät 2 (EtherCAT)^Klemme 1 (EK1200)^Klemme 3 (EL3446)^DPM Data^Data 12'}
	MDP5001_342_DPM_Data_Data_12_1					AT%Q* : UDINT;
	{attribute 'TcLinkTo' := 'TIID^Gerät 2 (EtherCAT)^Klemme 1 (EK1200)^Klemme 3 (EL3446)^DPM Data^Data 13'}
	MDP5001_342_DPM_Data_Data_13_1					AT%Q* : UDINT;
	{attribute 'TcLinkTo' := 'TIID^Gerät 2 (EtherCAT)^Klemme 1 (EK1200)^Klemme 3 (EL3446)^DPM Data^Data 14'}
	MDP5001_342_DPM_Data_Data_14_1					AT%Q* : UDINT;
	{attribute 'TcLinkTo' := 'TIID^Gerät 2 (EtherCAT)^Klemme 1 (EK1200)^Klemme 3 (EL3446)^DPM Data^Data 15'}
	MDP5001_342_DPM_Data_Data_15_1					AT%Q* : UDINT;
	{attribute 'TcLinkTo' := 'TIID^Gerät 2 (EtherCAT)^Klemme 1 (EK1200)^Klemme 3 (EL3446)^DPM Data^Data 16'}
	MDP5001_342_DPM_Data_Data_16_1					AT%Q* : UDINT;
	{attribute 'TcLinkTo' := 'TIID^Gerät 2 (EtherCAT)^Klemme 1 (EK1200)^Klemme 3 (EL3446)^DPM Data^Data 17'}
	MDP5001_342_DPM_Data_Data_17_1					AT%Q* : UDINT;
	{attribute 'TcLinkTo' := 'TIID^Gerät 2 (EtherCAT)^Klemme 1 (EK1200)^Klemme 3 (EL3446)^DPM Data^Data 18'}
	MDP5001_342_DPM_Data_Data_18_1					AT%Q* : UDINT;
	{attribute 'TcLinkTo' := 'TIID^Gerät 2 (EtherCAT)^Klemme 1 (EK1200)^Klemme 3 (EL3446)^DPM Data^Data 19'}
	MDP5001_342_DPM_Data_Data_19_1					AT%Q* : UDINT;
	{attribute 'TcLinkTo' := 'TIID^Gerät 2 (EtherCAT)^Klemme 1 (EK1200)^Klemme 3 (EL3446)^DPM Data^Data 20'}
	MDP5001_342_DPM_Data_Data_20_1					AT%Q* : UDINT;



// IOs for EL3446
	{attribute 'TcLinkTo' := 'TIID^Gerät 2 (EtherCAT)^Klemme 1 (EK1200)^Klemme 4 (EL3446)^I1 Channel^Overcurrent'}
	MDP5001_342_I1_Channel_Overcurrent_2						AT%I*  : BOOL;
	{attribute 'TcLinkTo' := 'TIID^Gerät 2 (EtherCAT)^Klemme 1 (EK1200)^Klemme 4 (EL3446)^I1 Channel^Inaccurate Current'}
	MDP5001_342_I1_Channel_Inaccurate_Current_2				AT%I*  : BOOL;
	{attribute 'TcLinkTo' := 'TIID^Gerät 2 (EtherCAT)^Klemme 1 (EK1200)^Klemme 4 (EL3446)^I1 Channel^Current Guard Warning'}
	MDP5001_342_I1_Channel_Current_Guard_Warning_2			AT%I*  : bool;
	{attribute 'TcLinkTo' := 'TIID^Gerät 2 (EtherCAT)^Klemme 1 (EK1200)^Klemme 4 (EL3446)^I1 Channel^Current Guard Error'}
	MDP5001_342_I1_Channel_Current_Guard_Error_2				AT%I*  : bool;
	{attribute 'TcLinkTo' := 'TIID^Gerät 2 (EtherCAT)^Klemme 1 (EK1200)^Klemme 4 (EL3446)^I1 Channel^Apparent Power Guard Warning'}
	MDP5001_342_I1_Channel_Apparent_Power_Guard_Warning_2		AT%I*  : bool;
	{attribute 'TcLinkTo' := 'TIID^Gerät 2 (EtherCAT)^Klemme 1 (EK1200)^Klemme 4 (EL3446)^I1 Channel^Apparent Power Guard Error'}
	MDP5001_342_I1_Channel_Apparent_Power_Guard_Error_2		AT%I*  : bool;
	{attribute 'TcLinkTo' := 'TIID^Gerät 2 (EtherCAT)^Klemme 1 (EK1200)^Klemme 4 (EL3446)^I1 Channel^Active Power Guard Warning'}
	MDP5001_342_I1_Channel_Active_Power_Guard_Warning_2		AT%I*  : bool;
	{attribute 'TcLinkTo' := 'TIID^Gerät 2 (EtherCAT)^Klemme 1 (EK1200)^Klemme 4 (EL3446)^I1 Channel^Active Power Guard Error'}
	MDP5001_342_I1_Channel_Active_Power_Guard_Error_2			AT%I*  : bool;
	{attribute 'TcLinkTo' := 'TIID^Gerät 2 (EtherCAT)^Klemme 1 (EK1200)^Klemme 4 (EL3446)^I1 Channel^Reactive Power Guard Warning'}
	MDP5001_342_I1_Channel_Reactive_Power_Guard_Warning_2		AT%I*  : bool;
	{attribute 'TcLinkTo' := 'TIID^Gerät 2 (EtherCAT)^Klemme 1 (EK1200)^Klemme 4 (EL3446)^I1 Channel^Reactive Power Guard Error'}
	MDP5001_342_I1_Channel_Reactive_Power_Guard_Error_2		AT%I*  : bool;
	{attribute 'TcLinkTo' := 'TIID^Gerät 2 (EtherCAT)^Klemme 1 (EK1200)^Klemme 4 (EL3446)^I1 Channel^DPM Inaccurate'}
	MDP5001_342_I1_Channel_DPM_Inaccurate_2					AT%I*  : bool;
	{attribute 'TcLinkTo' := 'TIID^Gerät 2 (EtherCAT)^Klemme 1 (EK1200)^Klemme 4 (EL3446)^I1 Channel^DPM Timeout'}
	MDP5001_342_I1_Channel_DPM_Timeout_2						AT%I*  : bool;
	{attribute 'TcLinkTo' := 'TIID^Gerät 2 (EtherCAT)^Klemme 1 (EK1200)^Klemme 4 (EL3446)^I1 Channel^TxPDO Toggle'}
	MDP5001_342_I1_Channel_TxPDO_Toggle_2						AT%I*  : bool;
	{attribute 'TcLinkTo' := 'TIID^Gerät 2 (EtherCAT)^Klemme 1 (EK1200)^Klemme 4 (EL3446)^I1 Channel^Current'}
	MDP5001_342_I1_Channel_Current_2							AT%I*  : REAL;
	{attribute 'TcLinkTo' := 'TIID^Gerät 2 (EtherCAT)^Klemme 1 (EK1200)^Klemme 4 (EL3446)^I1 Channel^Active Power'}
	MDP5001_342_I1_Channel_Active_Power_2						AT%I*  : REAL;
	{attribute 'TcLinkTo' := 'TIID^Gerät 2 (EtherCAT)^Klemme 1 (EK1200)^Klemme 4 (EL3446)^I1 Channel^Apparent Power'}
	MDP5001_342_I1_Channel_Apparent_Power_2					AT%I*  : REAL;
	{attribute 'TcLinkTo' := 'TIID^Gerät 2 (EtherCAT)^Klemme 1 (EK1200)^Klemme 4 (EL3446)^I1 Channel^Reactive Power Fundamental'}
	MDP5001_342_I1_Channel_Reactive_Power_Fundamental_2		AT%I*  : REAL;
	{attribute 'TcLinkTo' := 'TIID^Gerät 2 (EtherCAT)^Klemme 1 (EK1200)^Klemme 4 (EL3446)^I1 Channel^Active Energy'}
	MDP5001_342_I1_Channel_Active_Energy_2					AT%I*  : DINT;
	{attribute 'TcLinkTo' := 'TIID^Gerät 2 (EtherCAT)^Klemme 1 (EK1200)^Klemme 4 (EL3446)^I2 Channel^Overcurrent'}
	MDP5001_342_I2_Channel_Overcurrent_2						AT%I*  : BOOL;
	{attribute 'TcLinkTo' := 'TIID^Gerät 2 (EtherCAT)^Klemme 1 (EK1200)^Klemme 4 (EL3446)^I2 Channel^Inaccurate Current'}
	MDP5001_342_I2_Channel_Inaccurate_Current_2				AT%I*  : BOOL;
	{attribute 'TcLinkTo' := 'TIID^Gerät 2 (EtherCAT)^Klemme 1 (EK1200)^Klemme 4 (EL3446)^I2 Channel^Current Guard Warning'}
	MDP5001_342_I2_Channel_Current_Guard_Warning_2			AT%I*  : bool;
	{attribute 'TcLinkTo' := 'TIID^Gerät 2 (EtherCAT)^Klemme 1 (EK1200)^Klemme 4 (EL3446)^I2 Channel^Current Guard Error'}
	MDP5001_342_I2_Channel_Current_Guard_Error_2				AT%I*  : bool;
	{attribute 'TcLinkTo' := 'TIID^Gerät 2 (EtherCAT)^Klemme 1 (EK1200)^Klemme 4 (EL3446)^I2 Channel^Apparent Power Guard Warning'}
	MDP5001_342_I2_Channel_Apparent_Power_Guard_Warning_2		AT%I*  : bool;
	{attribute 'TcLinkTo' := 'TIID^Gerät 2 (EtherCAT)^Klemme 1 (EK1200)^Klemme 4 (EL3446)^I2 Channel^Apparent Power Guard Error'}
	MDP5001_342_I2_Channel_Apparent_Power_Guard_Error_2		AT%I*  : bool;
	{attribute 'TcLinkTo' := 'TIID^Gerät 2 (EtherCAT)^Klemme 1 (EK1200)^Klemme 4 (EL3446)^I2 Channel^Active Power Guard Warning'}
	MDP5001_342_I2_Channel_Active_Power_Guard_Warning_2		AT%I*  : bool;
	{attribute 'TcLinkTo' := 'TIID^Gerät 2 (EtherCAT)^Klemme 1 (EK1200)^Klemme 4 (EL3446)^I2 Channel^Active Power Guard Error'}
	MDP5001_342_I2_Channel_Active_Power_Guard_Error_2			AT%I*  : bool;
	{attribute 'TcLinkTo' := 'TIID^Gerät 2 (EtherCAT)^Klemme 1 (EK1200)^Klemme 4 (EL3446)^I2 Channel^Reactive Power Guard Warning'}
	MDP5001_342_I2_Channel_Reactive_Power_Guard_Warning_2		AT%I*  : bool;
	{attribute 'TcLinkTo' := 'TIID^Gerät 2 (EtherCAT)^Klemme 1 (EK1200)^Klemme 4 (EL3446)^I2 Channel^Reactive Power Guard Error'}
	MDP5001_342_I2_Channel_Reactive_Power_Guard_Error_2		AT%I*  : bool;
	{attribute 'TcLinkTo' := 'TIID^Gerät 2 (EtherCAT)^Klemme 1 (EK1200)^Klemme 4 (EL3446)^I2 Channel^DPM Inaccurate'}
	MDP5001_342_I2_Channel_DPM_Inaccurate_2					AT%I*  : bool;
	{attribute 'TcLinkTo' := 'TIID^Gerät 2 (EtherCAT)^Klemme 1 (EK1200)^Klemme 4 (EL3446)^I2 Channel^DPM Timeout'}
	MDP5001_342_I2_Channel_DPM_Timeout_2						AT%I*  : bool;
	{attribute 'TcLinkTo' := 'TIID^Gerät 2 (EtherCAT)^Klemme 1 (EK1200)^Klemme 4 (EL3446)^I2 Channel^TxPDO Toggle'}
	MDP5001_342_I2_Channel_TxPDO_Toggle_2						AT%I*  : bool;
	{attribute 'TcLinkTo' := 'TIID^Gerät 2 (EtherCAT)^Klemme 1 (EK1200)^Klemme 4 (EL3446)^I2 Channel^Current'}
	MDP5001_342_I2_Channel_Current_2							AT%I*  : REAL;
	{attribute 'TcLinkTo' := 'TIID^Gerät 2 (EtherCAT)^Klemme 1 (EK1200)^Klemme 4 (EL3446)^I2 Channel^Active Power'}
	MDP5001_342_I2_Channel_Active_Power_2						AT%I*  : REAL;
	{attribute 'TcLinkTo' := 'TIID^Gerät 2 (EtherCAT)^Klemme 1 (EK1200)^Klemme 4 (EL3446)^I2 Channel^Apparent Power'}
	MDP5001_342_I2_Channel_Apparent_Power_2					AT%I*  : REAL;
	{attribute 'TcLinkTo' := 'TIID^Gerät 2 (EtherCAT)^Klemme 1 (EK1200)^Klemme 4 (EL3446)^I2 Channel^Reactive Power Fundamental'}
	MDP5001_342_I2_Channel_Reactive_Power_Fundamental_2		AT%I*  : REAL;
	{attribute 'TcLinkTo' := 'TIID^Gerät 2 (EtherCAT)^Klemme 1 (EK1200)^Klemme 4 (EL3446)^I2 Channel^Active Energy'}
	MDP5001_342_I2_Channel_Active_Energy_2					AT%I*  : DINT;
	{attribute 'TcLinkTo' := 'TIID^Gerät 2 (EtherCAT)^Klemme 1 (EK1200)^Klemme 4 (EL3446)^I3 Channel^Overcurrent'}
	MDP5001_342_I3_Channel_Overcurrent_2						AT%I*  : BOOL;
	{attribute 'TcLinkTo' := 'TIID^Gerät 2 (EtherCAT)^Klemme 1 (EK1200)^Klemme 4 (EL3446)^I3 Channel^Inaccurate Current'}
	MDP5001_342_I3_Channel_Inaccurate_Current_2				AT%I*  : BOOL;
	{attribute 'TcLinkTo' := 'TIID^Gerät 2 (EtherCAT)^Klemme 1 (EK1200)^Klemme 4 (EL3446)^I3 Channel^Current Guard Warning'}
	MDP5001_342_I3_Channel_Current_Guard_Warning_2			AT%I*  : bool;
	{attribute 'TcLinkTo' := 'TIID^Gerät 2 (EtherCAT)^Klemme 1 (EK1200)^Klemme 4 (EL3446)^I3 Channel^Current Guard Error'}
	MDP5001_342_I3_Channel_Current_Guard_Error_2				AT%I*  : bool;
	{attribute 'TcLinkTo' := 'TIID^Gerät 2 (EtherCAT)^Klemme 1 (EK1200)^Klemme 4 (EL3446)^I3 Channel^Apparent Power Guard Warning'}
	MDP5001_342_I3_Channel_Apparent_Power_Guard_Warning_2		AT%I*  : bool;
	{attribute 'TcLinkTo' := 'TIID^Gerät 2 (EtherCAT)^Klemme 1 (EK1200)^Klemme 4 (EL3446)^I3 Channel^Apparent Power Guard Error'}
	MDP5001_342_I3_Channel_Apparent_Power_Guard_Error_2		AT%I*  : bool;
	{attribute 'TcLinkTo' := 'TIID^Gerät 2 (EtherCAT)^Klemme 1 (EK1200)^Klemme 4 (EL3446)^I3 Channel^Active Power Guard Warning'}
	MDP5001_342_I3_Channel_Active_Power_Guard_Warning_2		AT%I*  : bool;
	{attribute 'TcLinkTo' := 'TIID^Gerät 2 (EtherCAT)^Klemme 1 (EK1200)^Klemme 4 (EL3446)^I3 Channel^Active Power Guard Error'}
	MDP5001_342_I3_Channel_Active_Power_Guard_Error_2		AT%I*  : bool;
	{attribute 'TcLinkTo' := 'TIID^Gerät 2 (EtherCAT)^Klemme 1 (EK1200)^Klemme 4 (EL3446)^I3 Channel^Reactive Power Guard Warning'}
	MDP5001_342_I3_Channel_Reactive_Power_Guard_Warning_2		AT%I*  : bool;
	{attribute 'TcLinkTo' := 'TIID^Gerät 2 (EtherCAT)^Klemme 1 (EK1200)^Klemme 4 (EL3446)^I3 Channel^Reactive Power Guard Error'}
	MDP5001_342_I3_Channel_Reactive_Power_Guard_Error_2		AT%I*  : bool;
	{attribute 'TcLinkTo' := 'TIID^Gerät 2 (EtherCAT)^Klemme 1 (EK1200)^Klemme 4 (EL3446)^I3 Channel^DPM Inaccurate'}
	MDP5001_342_I3_Channel_DPM_Inaccurate_2					AT%I*  : bool;
	{attribute 'TcLinkTo' := 'TIID^Gerät 2 (EtherCAT)^Klemme 1 (EK1200)^Klemme 4 (EL3446)^I3 Channel^DPM Timeout'}
	MDP5001_342_I3_Channel_DPM_Timeout_2						AT%I*  : bool;
	{attribute 'TcLinkTo' := 'TIID^Gerät 2 (EtherCAT)^Klemme 1 (EK1200)^Klemme 4 (EL3446)^I3 Channel^TxPDO Toggle'}
	MDP5001_342_I3_Channel_TxPDO_Toggle_2						AT%I*  : bool;
	{attribute 'TcLinkTo' := 'TIID^Gerät 2 (EtherCAT)^Klemme 1 (EK1200)^Klemme 4 (EL3446)^I3 Channel^Current'}
	MDP5001_342_I3_Channel_Current_2							AT%I*  : REAL;
	{attribute 'TcLinkTo' := 'TIID^Gerät 2 (EtherCAT)^Klemme 1 (EK1200)^Klemme 4 (EL3446)^I3 Channel^Active Power'}
	MDP5001_342_I3_Channel_Active_Power_2						AT%I*  : REAL;
	{attribute 'TcLinkTo' := 'TIID^Gerät 2 (EtherCAT)^Klemme 1 (EK1200)^Klemme 4 (EL3446)^I3 Channel^Apparent Power'}
	MDP5001_342_I3_Channel_Apparent_Power_2					AT%I*  : REAL;
	{attribute 'TcLinkTo' := 'TIID^Gerät 2 (EtherCAT)^Klemme 1 (EK1200)^Klemme 4 (EL3446)^I3 Channel^Reactive Power Fundamental'}
	MDP5001_342_I3_Channel_Reactive_Power_Fundamental_2		AT%I*  : REAL;
	{attribute 'TcLinkTo' := 'TIID^Gerät 2 (EtherCAT)^Klemme 1 (EK1200)^Klemme 4 (EL3446)^I3 Channel^Active Energy'}
	MDP5001_342_I3_Channel_Active_Energy_2					AT%I*  : DINT;	
	{attribute 'TcLinkTo' := 'TIID^Gerät 2 (EtherCAT)^Klemme 1 (EK1200)^Klemme 4 (EL3446)^I4 Channel^Overcurrent'}
	MDP5001_342_I4_Channel_Overcurrent_2						AT%I*  : BOOL;
	{attribute 'TcLinkTo' := 'TIID^Gerät 2 (EtherCAT)^Klemme 1 (EK1200)^Klemme 4 (EL3446)^I4 Channel^Inaccurate Current'}
	MDP5001_342_I4_Channel_Inaccurate_Current_2				AT%I*  : BOOL;
	{attribute 'TcLinkTo' := 'TIID^Gerät 2 (EtherCAT)^Klemme 1 (EK1200)^Klemme 4 (EL3446)^I4 Channel^Current Guard Warning'}
	MDP5001_342_I4_Channel_Current_Guard_Warning_2			AT%I*  : bool;
	{attribute 'TcLinkTo' := 'TIID^Gerät 2 (EtherCAT)^Klemme 1 (EK1200)^Klemme 4 (EL3446)^I4 Channel^Current Guard Error'}
	MDP5001_342_I4_Channel_Current_Guard_Error_2				AT%I*  : bool;
	{attribute 'TcLinkTo' := 'TIID^Gerät 2 (EtherCAT)^Klemme 1 (EK1200)^Klemme 4 (EL3446)^I4 Channel^Apparent Power Guard Warning'}
	MDP5001_342_I4_Channel_Apparent_Power_Guard_Warning_2		AT%I*  : bool;
	{attribute 'TcLinkTo' := 'TIID^Gerät 2 (EtherCAT)^Klemme 1 (EK1200)^Klemme 4 (EL3446)^I4 Channel^Apparent Power Guard Error'}
	MDP5001_342_I4_Channel_Apparent_Power_Guard_Error_2		AT%I*  : bool;
	{attribute 'TcLinkTo' := 'TIID^Gerät 2 (EtherCAT)^Klemme 1 (EK1200)^Klemme 4 (EL3446)^I4 Channel^Active Power Guard Warning'}
	MDP5001_342_I4_Channel_Active_Power_Guard_Warning_2		AT%I*  : bool;
	{attribute 'TcLinkTo' := 'TIID^Gerät 2 (EtherCAT)^Klemme 1 (EK1200)^Klemme 4 (EL3446)^I4 Channel^Active Power Guard Error'}
	MDP5001_342_I4_Channel_Active_Power_Guard_Error_2			AT%I*  : bool;
	{attribute 'TcLinkTo' := 'TIID^Gerät 2 (EtherCAT)^Klemme 1 (EK1200)^Klemme 4 (EL3446)^I4 Channel^Reactive Power Guard Warning'}
	MDP5001_342_I4_Channel_Reactive_Power_Guard_Warning_2		AT%I*  : bool;
	{attribute 'TcLinkTo' := 'TIID^Gerät 2 (EtherCAT)^Klemme 1 (EK1200)^Klemme 4 (EL3446)^I4 Channel^Reactive Power Guard Error'}
	MDP5001_342_I4_Channel_Reactive_Power_Guard_Error_2		AT%I*  : bool;
	{attribute 'TcLinkTo' := 'TIID^Gerät 2 (EtherCAT)^Klemme 1 (EK1200)^Klemme 4 (EL3446)^I4 Channel^DPM Inaccurate'}
	MDP5001_342_I4_Channel_DPM_Inaccurate_2					AT%I*  : bool;
	{attribute 'TcLinkTo' := 'TIID^Gerät 2 (EtherCAT)^Klemme 1 (EK1200)^Klemme 4 (EL3446)^I4 Channel^DPM Timeout'}
	MDP5001_342_I4_Channel_DPM_Timeout_2						AT%I*  : bool;
	{attribute 'TcLinkTo' := 'TIID^Gerät 2 (EtherCAT)^Klemme 1 (EK1200)^Klemme 4 (EL3446)^I4 Channel^TxPDO Toggle'}
	MDP5001_342_I4_Channel_TxPDO_Toggle_2						AT%I*  : bool;
	{attribute 'TcLinkTo' := 'TIID^Gerät 2 (EtherCAT)^Klemme 1 (EK1200)^Klemme 4 (EL3446)^I4 Channel^Current'}
	MDP5001_342_I4_Channel_Current_2							AT%I*  : REAL;
	{attribute 'TcLinkTo' := 'TIID^Gerät 2 (EtherCAT)^Klemme 1 (EK1200)^Klemme 4 (EL3446)^I4 Channel^Active Power'}
	MDP5001_342_I4_Channel_Active_Power_2						AT%I*  : REAL;
	{attribute 'TcLinkTo' := 'TIID^Gerät 2 (EtherCAT)^Klemme 1 (EK1200)^Klemme 4 (EL3446)^I4 Channel^Apparent Power'}
	MDP5001_342_I4_Channel_Apparent_Power_2					AT%I*  : REAL;
	{attribute 'TcLinkTo' := 'TIID^Gerät 2 (EtherCAT)^Klemme 1 (EK1200)^Klemme 4 (EL3446)^I4 Channel^Reactive Power Fundamental'}
	MDP5001_342_I4_Channel_Reactive_Power_Fundamental_2		AT%I*  : REAL;
	{attribute 'TcLinkTo' := 'TIID^Gerät 2 (EtherCAT)^Klemme 1 (EK1200)^Klemme 4 (EL3446)^I4 Channel^Active Energy'}
	MDP5001_342_I4_Channel_Active_Energy_2					AT%I*  : DINT;
	{attribute 'TcLinkTo' := 'TIID^Gerät 2 (EtherCAT)^Klemme 1 (EK1200)^Klemme 4 (EL3446)^I5 Channel^Overcurrent'}
	MDP5001_342_I5_Channel_Overcurrent_2						AT%I*  : BOOL;
	{attribute 'TcLinkTo' := 'TIID^Gerät 2 (EtherCAT)^Klemme 1 (EK1200)^Klemme 4 (EL3446)^I5 Channel^Inaccurate Current'}
	MDP5001_342_I5_Channel_Inaccurate_Current_2				AT%I*  : BOOL;
	{attribute 'TcLinkTo' := 'TIID^Gerät 2 (EtherCAT)^Klemme 1 (EK1200)^Klemme 4 (EL3446)^I5 Channel^Current Guard Warning'}
	MDP5001_342_I5_Channel_Current_Guard_Warning_2			AT%I*  : bool;
	{attribute 'TcLinkTo' := 'TIID^Gerät 2 (EtherCAT)^Klemme 1 (EK1200)^Klemme 4 (EL3446)^I5 Channel^Current Guard Error'}
	MDP5001_342_I5_Channel_Current_Guard_Error_2				AT%I*  : bool;
	{attribute 'TcLinkTo' := 'TIID^Gerät 2 (EtherCAT)^Klemme 1 (EK1200)^Klemme 4 (EL3446)^I5 Channel^Apparent Power Guard Warning'}
	MDP5001_342_I5_Channel_Apparent_Power_Guard_Warning_2		AT%I*  : bool;
	{attribute 'TcLinkTo' := 'TIID^Gerät 2 (EtherCAT)^Klemme 1 (EK1200)^Klemme 4 (EL3446)^I5 Channel^Apparent Power Guard Error'}
	MDP5001_342_I5_Channel_Apparent_Power_Guard_Error_2		AT%I*  : bool;
	{attribute 'TcLinkTo' := 'TIID^Gerät 2 (EtherCAT)^Klemme 1 (EK1200)^Klemme 4 (EL3446)^I5 Channel^Active Power Guard Warning'}
	MDP5001_342_I5_Channel_Active_Power_Guard_Warning_2		AT%I*  : bool;
	{attribute 'TcLinkTo' := 'TIID^Gerät 2 (EtherCAT)^Klemme 1 (EK1200)^Klemme 4 (EL3446)^I5 Channel^Active Power Guard Error'}
	MDP5001_342_I5_Channel_Active_Power_Guard_Error_2			AT%I*  : bool;
	{attribute 'TcLinkTo' := 'TIID^Gerät 2 (EtherCAT)^Klemme 1 (EK1200)^Klemme 4 (EL3446)^I5 Channel^Reactive Power Guard Warning'}
	MDP5001_342_I5_Channel_Reactive_Power_Guard_Warning_2		AT%I*  : bool;
	{attribute 'TcLinkTo' := 'TIID^Gerät 2 (EtherCAT)^Klemme 1 (EK1200)^Klemme 4 (EL3446)^I5 Channel^Reactive Power Guard Error'}
	MDP5001_342_I5_Channel_Reactive_Power_Guard_Error_2		AT%I*  : bool;
	{attribute 'TcLinkTo' := 'TIID^Gerät 2 (EtherCAT)^Klemme 1 (EK1200)^Klemme 4 (EL3446)^I5 Channel^DPM Inaccurate'}
	MDP5001_342_I5_Channel_DPM_Inaccurate_2					AT%I*  : bool;
	{attribute 'TcLinkTo' := 'TIID^Gerät 2 (EtherCAT)^Klemme 1 (EK1200)^Klemme 4 (EL3446)^I5 Channel^DPM Timeout'}
	MDP5001_342_I5_Channel_DPM_Timeout_2						AT%I*  : bool;
	{attribute 'TcLinkTo' := 'TIID^Gerät 2 (EtherCAT)^Klemme 1 (EK1200)^Klemme 4 (EL3446)^I5 Channel^TxPDO Toggle'}
	MDP5001_342_I5_Channel_TxPDO_Toggle_2						AT%I*  : bool;
	{attribute 'TcLinkTo' := 'TIID^Gerät 2 (EtherCAT)^Klemme 1 (EK1200)^Klemme 4 (EL3446)^I5 Channel^Current'}
	MDP5001_342_I5_Channel_Current_2							AT%I*  : REAL;
	{attribute 'TcLinkTo' := 'TIID^Gerät 2 (EtherCAT)^Klemme 1 (EK1200)^Klemme 4 (EL3446)^I5 Channel^Active Power'}
	MDP5001_342_I5_Channel_Active_Power_2						AT%I*  : REAL;
	{attribute 'TcLinkTo' := 'TIID^Gerät 2 (EtherCAT)^Klemme 1 (EK1200)^Klemme 4 (EL3446)^I5 Channel^Apparent Power'}
	MDP5001_342_I5_Channel_Apparent_Power_2					AT%I*  : REAL;
	{attribute 'TcLinkTo' := 'TIID^Gerät 2 (EtherCAT)^Klemme 1 (EK1200)^Klemme 4 (EL3446)^I5 Channel^Reactive Power Fundamental'}
	MDP5001_342_I5_Channel_Reactive_Power_Fundamental_2		AT%I*  : REAL;
	{attribute 'TcLinkTo' := 'TIID^Gerät 2 (EtherCAT)^Klemme 1 (EK1200)^Klemme 4 (EL3446)^I5 Channel^Active Energy'}
	MDP5001_342_I5_Channel_Active_Energy_2					AT%I*  : DINT;
	{attribute 'TcLinkTo' := 'TIID^Gerät 2 (EtherCAT)^Klemme 1 (EK1200)^Klemme 4 (EL3446)^I6 Channel^Overcurrent'}
	MDP5001_342_I6_Channel_Overcurrent_2						AT%I*  : BOOL;
	{attribute 'TcLinkTo' := 'TIID^Gerät 2 (EtherCAT)^Klemme 1 (EK1200)^Klemme 4 (EL3446)^I6 Channel^Inaccurate Current'}
	MDP5001_342_I6_Channel_Inaccurate_Current_2				AT%I*  : BOOL;
	{attribute 'TcLinkTo' := 'TIID^Gerät 2 (EtherCAT)^Klemme 1 (EK1200)^Klemme 4 (EL3446)^I6 Channel^Current Guard Warning'}
	MDP5001_342_I6_Channel_Current_Guard_Warning_2			AT%I*  : bool;
	{attribute 'TcLinkTo' := 'TIID^Gerät 2 (EtherCAT)^Klemme 1 (EK1200)^Klemme 4 (EL3446)^I6 Channel^Current Guard Error'}
	MDP5001_342_I6_Channel_Current_Guard_Error_2				AT%I*  : bool;
	{attribute 'TcLinkTo' := 'TIID^Gerät 2 (EtherCAT)^Klemme 1 (EK1200)^Klemme 4 (EL3446)^I6 Channel^Apparent Power Guard Warning'}
	MDP5001_342_I6_Channel_Apparent_Power_Guard_Warning_2		AT%I*  : bool;
	{attribute 'TcLinkTo' := 'TIID^Gerät 2 (EtherCAT)^Klemme 1 (EK1200)^Klemme 4 (EL3446)^I6 Channel^Apparent Power Guard Error'}
	MDP5001_342_I6_Channel_Apparent_Power_Guard_Error_2		AT%I*  : bool;
	{attribute 'TcLinkTo' := 'TIID^Gerät 2 (EtherCAT)^Klemme 1 (EK1200)^Klemme 4 (EL3446)^I6 Channel^Active Power Guard Warning'}
	MDP5001_342_I6_Channel_Active_Power_Guard_Warning_2		AT%I*  : bool;
	{attribute 'TcLinkTo' := 'TIID^Gerät 2 (EtherCAT)^Klemme 1 (EK1200)^Klemme 4 (EL3446)^I6 Channel^Active Power Guard Error'}
	MDP5001_342_I6_Channel_Active_Power_Guard_Error_2			AT%I*  : bool;
	{attribute 'TcLinkTo' := 'TIID^Gerät 2 (EtherCAT)^Klemme 1 (EK1200)^Klemme 4 (EL3446)^I6 Channel^Reactive Power Guard Warning'}
	MDP5001_342_I6_Channel_Reactive_Power_Guard_Warning_2		AT%I*  : bool;
	{attribute 'TcLinkTo' := 'TIID^Gerät 2 (EtherCAT)^Klemme 1 (EK1200)^Klemme 4 (EL3446)^I6 Channel^Reactive Power Guard Error'}
	MDP5001_342_I6_Channel_Reactive_Power_Guard_Error_2		AT%I*  : bool;
	{attribute 'TcLinkTo' := 'TIID^Gerät 2 (EtherCAT)^Klemme 1 (EK1200)^Klemme 4 (EL3446)^I6 Channel^DPM Inaccurate'}
	MDP5001_342_I6_Channel_DPM_Inaccurate_2					AT%I*  : bool;
	{attribute 'TcLinkTo' := 'TIID^Gerät 2 (EtherCAT)^Klemme 1 (EK1200)^Klemme 4 (EL3446)^I6 Channel^DPM Timeout'}
	MDP5001_342_I6_Channel_DPM_Timeout_2						AT%I*  : bool;
	{attribute 'TcLinkTo' := 'TIID^Gerät 2 (EtherCAT)^Klemme 1 (EK1200)^Klemme 4 (EL3446)^I6 Channel^TxPDO Toggle'}
	MDP5001_342_I6_Channel_TxPDO_Toggle_2						AT%I*  : bool;
	{attribute 'TcLinkTo' := 'TIID^Gerät 2 (EtherCAT)^Klemme 1 (EK1200)^Klemme 4 (EL3446)^I6 Channel^Current'}
	MDP5001_342_I6_Channel_Current_2							AT%I*  : REAL;
	{attribute 'TcLinkTo' := 'TIID^Gerät 2 (EtherCAT)^Klemme 1 (EK1200)^Klemme 4 (EL3446)^I6 Channel^Active Power'}
	MDP5001_342_I6_Channel_Active_Power_2						AT%I*  : REAL;
	{attribute 'TcLinkTo' := 'TIID^Gerät 2 (EtherCAT)^Klemme 1 (EK1200)^Klemme 4 (EL3446)^I6 Channel^Apparent Power'}
	MDP5001_342_I6_Channel_Apparent_Power_2					AT%I*  : REAL;
	{attribute 'TcLinkTo' := 'TIID^Gerät 2 (EtherCAT)^Klemme 1 (EK1200)^Klemme 4 (EL3446)^I6 Channel^Reactive Power Fundamental'}
	MDP5001_342_I6_Channel_Reactive_Power_Fundamental_2		AT%I*  : REAL;
	{attribute 'TcLinkTo' := 'TIID^Gerät 2 (EtherCAT)^Klemme 1 (EK1200)^Klemme 4 (EL3446)^I6 Channel^Active Energy'}
	MDP5001_342_I6_Channel_Active_Energy_2					AT%I*  : DINT;	
	
	{attribute 'TcLinkTo' := 'TIID^Gerät 2 (EtherCAT)^Klemme 1 (EK1200)^Klemme 4 (EL3446)^DPM Variant Value In^TxPDO Toggle'}
	MDP5001_342_DPM_Variant_Value_In_TxPDO_Toggle_2			AT%I*  : BOOL;
	{attribute 'TcLinkTo' := 'TIID^Gerät 2 (EtherCAT)^Klemme 1 (EK1200)^Klemme 4 (EL3446)^DPM Variant Value In^Index 1 REAL'}
	MDP5001_342_DPM_Variant_Value_In_Index_1_REAL_2			AT%I*  : UINT;
	{attribute 'TcLinkTo' := 'TIID^Gerät 2 (EtherCAT)^Klemme 1 (EK1200)^Klemme 4 (EL3446)^DPM Variant Value In^Value 1 REAL'}
	MDP5001_342_DPM_Variant_Value_In_Value_1_REAL_2			AT%I*  : REAL;
	{attribute 'TcLinkTo' := 'TIID^Gerät 2 (EtherCAT)^Klemme 1 (EK1200)^Klemme 4 (EL3446)^DPM Variant Value In^Index 2 REAL'}
	MDP5001_342_DPM_Variant_Value_In_Index_2_REAL_2			AT%I*  : UINT;
	{attribute 'TcLinkTo' := 'TIID^Gerät 2 (EtherCAT)^Klemme 1 (EK1200)^Klemme 4 (EL3446)^DPM Variant Value In^Value 2 REAL'}
	MDP5001_342_DPM_Variant_Value_In_Value_2_REAL_2			AT%I*  : REAL;
	{attribute 'TcLinkTo' := 'TIID^Gerät 2 (EtherCAT)^Klemme 1 (EK1200)^Klemme 4 (EL3446)^DPM Variant Value In^Index 3 REAL'}
	MDP5001_342_DPM_Variant_Value_In_Index_3_REAL_2			AT%I*  : UINT;
	{attribute 'TcLinkTo' := 'TIID^Gerät 2 (EtherCAT)^Klemme 1 (EK1200)^Klemme 4 (EL3446)^DPM Variant Value In^Value 3 REAL'}
	MDP5001_342_DPM_Variant_Value_In_Value_3_REAL_2			AT%I*  : REAL;
	{attribute 'TcLinkTo' := 'TIID^Gerät 2 (EtherCAT)^Klemme 1 (EK1200)^Klemme 4 (EL3446)^DPM Variant Value In^Index 4 ULINT'}
	MDP5001_342_DPM_Variant_Value_In_Index_4_ULINT_2			AT%I*  : UINT;
	{attribute 'TcLinkTo' := 'TIID^Gerät 2 (EtherCAT)^Klemme 1 (EK1200)^Klemme 4 (EL3446)^DPM Variant Value In^Value 4 ULINT'}
	MDP5001_342_DPM_Variant_Value_In_Value_4_ULINT_2			AT%I*  : ULINT;

	{attribute 'TcLinkTo' := 'TIID^Gerät 2 (EtherCAT)^Klemme 1 (EK1200)^Klemme 4 (EL3446)^DPM Variant Value Out^Index 1 REAL'}
	MDP5001_342_DPM_Variant_Value_Out_Index_1_REAL_2	AT%Q* : UINT;
	{attribute 'TcLinkTo' := 'TIID^Gerät 2 (EtherCAT)^Klemme 1 (EK1200)^Klemme 4 (EL3446)^DPM Variant Value Out^Index 2 REAL'}
	MDP5001_342_DPM_Variant_Value_Out_Index_2_REAL_2	AT%Q* : UINT;
	{attribute 'TcLinkTo' := 'TIID^Gerät 2 (EtherCAT)^Klemme 1 (EK1200)^Klemme 4 (EL3446)^DPM Variant Value Out^Index 3 REAL'}
	MDP5001_342_DPM_Variant_Value_Out_Index_3_REAL_2	AT%Q* : UINT;
	{attribute 'TcLinkTo' := 'TIID^Gerät 2 (EtherCAT)^Klemme 1 (EK1200)^Klemme 4 (EL3446)^DPM Variant Value Out^Index 4 ULINT'}
	MDP5001_342_DPM_Variant_Value_Out_Index_4_ULINT_2	AT%Q* : UINT;
	{attribute 'TcLinkTo' := 'TIID^Gerät 2 (EtherCAT)^Klemme 1 (EK1200)^Klemme 4 (EL3446)^DPM Data^Data 1'}
	MDP5001_342_DPM_Data_Data_1_2						AT%Q* : UDINT;
	{attribute 'TcLinkTo' := 'TIID^Gerät 2 (EtherCAT)^Klemme 1 (EK1200)^Klemme 4 (EL3446)^DPM Data^Data 2'}
	MDP5001_342_DPM_Data_Data_2_2						AT%Q* : UDINT;
	{attribute 'TcLinkTo' := 'TIID^Gerät 2 (EtherCAT)^Klemme 1 (EK1200)^Klemme 4 (EL3446)^DPM Data^Data 3'}
	MDP5001_342_DPM_Data_Data_3_2						AT%Q* : UDINT;
	{attribute 'TcLinkTo' := 'TIID^Gerät 2 (EtherCAT)^Klemme 1 (EK1200)^Klemme 4 (EL3446)^DPM Data^Data 4'}
	MDP5001_342_DPM_Data_Data_4_2						AT%Q* : UDINT;
	{attribute 'TcLinkTo' := 'TIID^Gerät 2 (EtherCAT)^Klemme 1 (EK1200)^Klemme 4 (EL3446)^DPM Data^Data 5'}
	MDP5001_342_DPM_Data_Data_5_2						AT%Q* : UDINT;
	{attribute 'TcLinkTo' := 'TIID^Gerät 2 (EtherCAT)^Klemme 1 (EK1200)^Klemme 4 (EL3446)^DPM Data^Data 6'}
	MDP5001_342_DPM_Data_Data_6_2						AT%Q* : UDINT;
	{attribute 'TcLinkTo' := 'TIID^Gerät 2 (EtherCAT)^Klemme 1 (EK1200)^Klemme 4 (EL3446)^DPM Data^Data 7'}
	MDP5001_342_DPM_Data_Data_7_2						AT%Q* : UDINT;
	{attribute 'TcLinkTo' := 'TIID^Gerät 2 (EtherCAT)^Klemme 1 (EK1200)^Klemme 4 (EL3446)^DPM Data^Data 8'}
	MDP5001_342_DPM_Data_Data_8_2						AT%Q* : UDINT;
	{attribute 'TcLinkTo' := 'TIID^Gerät 2 (EtherCAT)^Klemme 1 (EK1200)^Klemme 4 (EL3446)^DPM Data^Data 9'}
	MDP5001_342_DPM_Data_Data_9_2						AT%Q* : UDINT;
	{attribute 'TcLinkTo' := 'TIID^Gerät 2 (EtherCAT)^Klemme 1 (EK1200)^Klemme 4 (EL3446)^DPM Data^Data 10'}
	MDP5001_342_DPM_Data_Data_10_2					AT%Q* : UDINT;
	{attribute 'TcLinkTo' := 'TIID^Gerät 2 (EtherCAT)^Klemme 1 (EK1200)^Klemme 4 (EL3446)^DPM Data^Data 11'}
	MDP5001_342_DPM_Data_Data_11_2					AT%Q* : UDINT;
	{attribute 'TcLinkTo' := 'TIID^Gerät 2 (EtherCAT)^Klemme 1 (EK1200)^Klemme 4 (EL3446)^DPM Data^Data 12'}
	MDP5001_342_DPM_Data_Data_12_2					AT%Q* : UDINT;
	{attribute 'TcLinkTo' := 'TIID^Gerät 2 (EtherCAT)^Klemme 1 (EK1200)^Klemme 4 (EL3446)^DPM Data^Data 13'}
	MDP5001_342_DPM_Data_Data_13_2					AT%Q* : UDINT;
	{attribute 'TcLinkTo' := 'TIID^Gerät 2 (EtherCAT)^Klemme 1 (EK1200)^Klemme 4 (EL3446)^DPM Data^Data 14'}
	MDP5001_342_DPM_Data_Data_14_2					AT%Q* : UDINT;
	{attribute 'TcLinkTo' := 'TIID^Gerät 2 (EtherCAT)^Klemme 1 (EK1200)^Klemme 4 (EL3446)^DPM Data^Data 15'}
	MDP5001_342_DPM_Data_Data_15_2					AT%Q* : UDINT;
	{attribute 'TcLinkTo' := 'TIID^Gerät 2 (EtherCAT)^Klemme 1 (EK1200)^Klemme 4 (EL3446)^DPM Data^Data 16'}
	MDP5001_342_DPM_Data_Data_16_2					AT%Q* : UDINT;
	{attribute 'TcLinkTo' := 'TIID^Gerät 2 (EtherCAT)^Klemme 1 (EK1200)^Klemme 4 (EL3446)^DPM Data^Data 17'}
	MDP5001_342_DPM_Data_Data_17_2					AT%Q* : UDINT;
	{attribute 'TcLinkTo' := 'TIID^Gerät 2 (EtherCAT)^Klemme 1 (EK1200)^Klemme 4 (EL3446)^DPM Data^Data 18'}
	MDP5001_342_DPM_Data_Data_18_2					AT%Q* : UDINT;
	{attribute 'TcLinkTo' := 'TIID^Gerät 2 (EtherCAT)^Klemme 1 (EK1200)^Klemme 4 (EL3446)^DPM Data^Data 19'}
	MDP5001_342_DPM_Data_Data_19_2					AT%Q* : UDINT;
	{attribute 'TcLinkTo' := 'TIID^Gerät 2 (EtherCAT)^Klemme 1 (EK1200)^Klemme 4 (EL3446)^DPM Data^Data 20'}
	MDP5001_342_DPM_Data_Data_20_2					AT%Q* : UDINT;

END_VAR

// copy HW Data to FBs accordingly
//EL3443

